LIN {X 0,Y 149.058,Z 383.574,A -85,B 0,C 180,E1 -25603.016,E2 -25603.016} C_VEL
LIN {X 0,Y 150.368,Z 387.947,A -85,B 0,C 180,E1 -25603.742,E2 -25603.742} C_VEL
LIN {X 0,Y 150.892,Z 399.258,A -85,B 0,C 180,E1 -25604.619,E2 -25604.619} C_VEL
LIN {X 0,Y 148.093,Z 440.283,A -85,B 0,C 180,E1 -25606.367,E2 -25606.367} C_VEL
LIN {X 0,Y 146.164,Z 454.102,A -85,B 0,C 180,E1 -25607.428,E2 -25607.428} C_VEL
LIN {X 0,Y 143.596,Z 466.563,A -85,B 0,C 180,E1 -25608.88,E2 -25608.88} C_VEL
LIN {X 0,Y 140.912,Z 476.802,A -85,B 0,C 180,E1 -25610.515,E2 -25610.515} C_VEL
LIN {X 0,Y 137.697,Z 487.195,A -85,B 0,C 180,E1 -25612.695,E2 -25612.695} C_VEL
LIN {X 0,Y 134.338,Z 496.866,A -85,B 0,C 180,E1 -25615.327,E2 -25615.327} C_VEL
LIN {X 0,Y 131.02,Z 505.835,A -85,B 0,C 180,E1 -25618.469,E2 -25618.469} C_VEL
LIN {X 0,Y 127.707,Z 513.721,A -85,B 0,C 180,E1 -25621.923,E2 -25621.923} C_VEL
LIN {X 0,Y 125.501,Z 519.623,A -85,B 0,C 180,E1 -25625.168,E2 -25625.168} C_VEL
LIN {X 0,Y 122.78,Z 526.537,A -85,B 0,C 180,E1 -25629.915,E2 -25629.915} C_VEL
LIN {X 0,Y 120.837,Z 532.058,A -85,B 0,C 180,E1 -25634.83,E2 -25634.83} C_VEL
LIN {X 0,Y 119.81,Z 536.375,A -85,B 0,C 180,E1 -25639.866,E2 -25639.866} C_VEL
LIN {X 0,Y 119.472,Z 538.652,A -85,B 0,C 180,E1 -25643.245,E2 -25643.245} C_VEL
LIN {X 0,Y 119.372,Z 540.456,A -85,B 0,C 180,E1 -25646.627,E2 -25646.627} C_VEL
LIN {X 0,Y 119.478,Z 541.86,A -85,B 0,C 180,E1 -25650.172,E2 -25650.172} C_VEL
LIN {X 0,Y 119.353,Z 542.729,A -85,B 0,C 180,E1 -25653.377,E2 -25653.377} C_VEL
LIN {X 0,Y 119.418,Z 543.262,A -85,B 0,C 180,E1 -25656.761,E2 -25656.761} C_VEL
LIN {X 0,Y 119.832,Z 543.392,A -85,B 0,C 180,E1 -25660.135,E2 -25660.135} C_VEL
LIN {X 0,Y 121.629,Z 542.443,A -85,B 0,C 180,E1 -25666.794,E2 -25666.794} C_VEL
LIN {X 0,Y 123.064,Z 541.401,A -85,B 0,C 180,E1 -25670.04,E2 -25670.04} C_VEL
LIN {X 0,Y 126.605,Z 538.614,A -85,B 0,C 180,E1 -25675.353,E2 -25675.353} C_VEL
LIN {X 0,Y 129.964,Z 535.757,A -85,B 0,C 180,E1 -25679.125,E2 -25679.125} C_VEL
LIN {X 0,Y 134.618,Z 531.251,A -85,B 0,C 180,E1 -25683.418,E2 -25683.418} C_VEL
LIN {X 0,Y 138.6,Z 526.986,A -85,B 0,C 180,E1 -25686.503,E2 -25686.503} C_VEL
LIN {X 0,Y 140.715,Z 524.056,A -85,B 0,C 180,E1 -25688.426,E2 -25688.426} C_VEL
LIN {X 0,Y 142.976,Z 518.943,A -85,B 0,C 180,E1 -25691.745,E2 -25691.745} C_VEL
LIN {X 0,Y 145.492,Z 513.259,A -85,B 0,C 180,E1 -25694.806,E2 -25694.806} C_VEL
LIN {X 0,Y 147.901,Z 509.417,A -85,B 0,C 180,E1 -25696.279,E2 -25696.279} C_VEL
LIN {X 0,Y 154.805,Z 499.219,A -85,B 0,C 180,E1 -25699.006,E2 -25699.006} C_VEL
LIN {X 0,Y 159.828,Z 490.367,A -85,B 0,C 180,E1 -25700.807,E2 -25700.807} C_VEL
LIN {X 0,Y 164.4,Z 481.018,A -85,B 0,C 180,E1 -25702.267,E2 -25702.267} C_VEL
LIN {X 0,Y 169.126,Z 469.344,A -85,B 0,C 180,E1 -25703.623,E2 -25703.623} C_VEL
LIN {X 0,Y 173.178,Z 456.095,A -85,B 0,C 180,E1 -25704.732,E2 -25704.732} C_VEL
LIN {X 0,Y 175.889,Z 443.42,A -85,B 0,C 180,E1 -25705.467,E2 -25705.467} C_VEL
LIN {X 0,Y 177.616,Z 429.252,A -85,B 0,C 180,E1 -25705.973,E2 -25705.973} C_VEL
LIN {X 0,Y 178.336,Z 420.642,A -85,B 0,C 180,E1 -25706.258,E2 -25706.258} C_VEL
LIN {X 0,Y 174.777,Z 410.912,A -85,B 0,C 180,E1 -25709.285,E2 -25709.285} C_VEL
LIN {X 0,Y 170.975,Z 401.854,A -85,B 0,C 180,E1 -25712.952,E2 -25712.952} C_VEL
LIN {X 0,Y 168.609,Z 396.773,A -85,B 0,C 180,E1 -25715.583,E2 -25715.583} C_VEL
LIN {X 0,Y 166.432,Z 392.274,A -85,B 0,C 180,E1 -25718.394,E2 -25718.394} C_VEL
LIN {X 0,Y 164.505,Z 389.028,A -85,B 0,C 180,E1 -25721.312,E2 -25721.312} C_VEL
LIN {X 0,Y 162.526,Z 386.151,A -85,B 0,C 180,E1 -25725.122,E2 -25725.122} C_VEL
LIN {X 0,Y 162.034,Z 384.768,A -85,B 0,C 180,E1 -25726.518,E2 -25726.518} C_VEL
LIN {X 0,Y 160.404,Z 383.082,A -85,B 0,C 180,E1 -25733.431,E2 -25733.431} C_VEL
LIN {X 0,Y 160.639,Z 382.941,A -85,B 0,C 180,E1 -25738.746,E2 -25738.746} C_VEL
LIN {X 0,Y 162.248,Z 384.816,A -85,B 0,C 180,E1 -25744.521,E2 -25744.521} C_VEL
LIN {X 0,Y 163.939,Z 388.212,A -85,B 0,C 180,E1 -25748.271,E2 -25748.271} C_VEL
LIN {X 0,Y 164.958,Z 389.595,A -85,B 0,C 180,E1 -25749.949,E2 -25749.949} C_VEL
LIN {X 0,Y 167.66,Z 394.12,A -85,B 0,C 180,E1 -25753.715,E2 -25753.715} C_VEL
LIN {X 0,Y 170.258,Z 398.497,A -85,B 0,C 180,E1 -25756.64,E2 -25756.64} C_VEL
LIN {X 0,Y 173.134,Z 403.391,A -85,B 0,C 180,E1 -25759.411,E2 -25759.411} C_VEL
LIN {X 0,Y 177.436,Z 411.732,A -85,B 0,C 180,E1 -25763.025,E2 -25763.025} C_VEL
LIN {X 0,Y 178.8,Z 414.577,A -85,B 0,C 180,E1 -25764.067,E2 -25764.067} C_VEL
LIN {X 0,Y 176.796,Z 434.165,A -85,B 0,C 180,E1 -25764.728,E2 -25764.728} C_VEL
LIN {X 0,Y 174.585,Z 446.23,A -85,B 0,C 180,E1 -25765.419,E2 -25765.419} C_VEL
LIN {X 0,Y 171.577,Z 457.31,A -85,B 0,C 180,E1 -25766.265,E2 -25766.265} C_VEL
LIN {X 0,Y 167.687,Z 468.926,A -85,B 0,C 180,E1 -25767.613,E2 -25767.613} C_VEL
LIN {X 0,Y 162.984,Z 479.606,A -85,B 0,C 180,E1 -25769.167,E2 -25769.167} C_VEL
LIN {X 0,Y 157.343,Z 490.399,A -85,B 0,C 180,E1 -25771.322,E2 -25771.322} C_VEL
LIN {X 0,Y 151.116,Z 500.294,A -85,B 0,C 180,E1 -25773.923,E2 -25773.923} C_VEL
LIN {X 0,Y 144.848,Z 508.604,A -85,B 0,C 180,E1 -25776.813,E2 -25776.813} C_VEL
LIN {X 0,Y 138.384,Z 516.119,A -85,B 0,C 180,E1 -25780.376,E2 -25780.376} C_VEL
LIN {X 0,Y 132.495,Z 522.113,A -85,B 0,C 180,E1 -25784.266,E2 -25784.266} C_VEL
LIN {X 0,Y 127.231,Z 526.808,A -85,B 0,C 180,E1 -25788.48,E2 -25788.48} C_VEL
LIN {X 0,Y 122.221,Z 530.713,A -85,B 0,C 180,E1 -25793.613,E2 -25793.613} C_VEL
LIN {X 0,Y 118.941,Z 532.846,A -85,B 0,C 180,E1 -25797.872,E2 -25797.872} C_VEL
LIN {X 0,Y 116.872,Z 533.975,A -85,B 0,C 180,E1 -25801.243,E2 -25801.243} C_VEL
LIN {X 0,Y 113.924,Z 534.95,A -85,B 0,C 180,E1 -25808.274,E2 -25808.274} C_VEL
LIN {X 0,Y 112.953,Z 534.852,A -85,B 0,C 180,E1 -25811.873,E2 -25811.873} C_VEL
LIN {X 0,Y 112.312,Z 534.327,A -85,B 0,C 180,E1 -25815.503,E2 -25815.503} C_VEL
LIN {X 0,Y 112.071,Z 533.382,A -85,B 0,C 180,E1 -25819.154,E2 -25819.154} C_VEL
LIN {X 0,Y 112.159,Z 532.044,A -85,B 0,C 180,E1 -25822.799,E2 -25822.799} C_VEL
LIN {X 0,Y 112.759,Z 529.463,A -85,B 0,C 180,E1 -25827.831,E2 -25827.831} C_VEL
LIN {X 0,Y 113.913,Z 525.425,A -85,B 0,C 180,E1 -25833.535,E2 -25833.535} C_VEL
LIN {X 0,Y 115.858,Z 520.489,A -85,B 0,C 180,E1 -25838.721,E2 -25838.721} C_VEL
LIN {X 0,Y 118.494,Z 514.292,A -85,B 0,C 180,E1 -25843.722,E2 -25843.722} C_VEL
LIN {X 0,Y 121.887,Z 506.562,A -85,B 0,C 180,E1 -25848.487,E2 -25848.487} C_VEL
LIN {X 0,Y 126,Z 496.881,A -85,B 0,C 180,E1 -25852.98,E2 -25852.98} C_VEL
LIN {X 0,Y 129.987,Z 486.863,A -85,B 0,C 180,E1 -25856.489,E2 -25856.489} C_VEL
LIN {X 0,Y 134.034,Z 475.483,A -85,B 0,C 180,E1 -25859.442,E2 -25859.442} C_VEL
LIN {X 0,Y 137.352,Z 464.338,A -85,B 0,C 180,E1 -25861.63,E2 -25861.63} C_VEL
LIN {X 0,Y 139.997,Z 452,A -85,B 0,C 180,E1 -25863.517,E2 -25863.517} C_VEL
LIN {X 0,Y 141.902,Z 439.97,A -85,B 0,C 180,E1 -25864.799,E2 -25864.799} C_VEL
LIN {X 0,Y 143.526,Z 426.582,A -85,B 0,C 180,E1 -25865.609,E2 -25865.609} C_VEL
LIN {X 0,Y 146.26,Z 386.175,A -85,B 0,C 180,E1 -25867.309,E2 -25867.309} C_VEL
LIN {X 0,Y 141.15,Z 375.197,A -85,B 0,C 180,E1 -25870.058,E2 -25870.058} C_VEL
LIN {X 0,Y 136.174,Z 366.246,A -85,B 0,C 180,E1 -25872.941,E2 -25872.941} C_VEL
LIN {X 0,Y 131.196,Z 358.517,A -85,B 0,C 180,E1 -25876.129,E2 -25876.129} C_VEL
LIN {X 0,Y 128.748,Z 355.059,A -85,B 0,C 180,E1 -25877.845,E2 -25877.845} C_VEL
LIN {X 0,Y 125.996,Z 351.155,A -85,B 0,C 180,E1 -25879.951,E2 -25879.951} C_VEL
LIN {X 0,Y 123.491,Z 347.657,A -85,B 0,C 180,E1 -25882.052,E2 -25882.052} C_VEL
LIN {X 0,Y 122.516,Z 346.611,A -85,B 0,C 180,E1 -25882.893,E2 -25882.893} C_VEL
LIN {X 0,Y 120.143,Z 343.788,A -85,B 0,C 180,E1 -25885.123,E2 -25885.123} C_VEL
LIN {X 0,Y 119.192,Z 341.849,A -85,B 0,C 180,E1 -25886.187,E2 -25886.187} C_VEL
LIN {X 0,Y 116.758,Z 340.164,A -85,B 0,C 180,E1 -25888.72,E2 -25888.72} C_VEL
LIN {X 0,Y 115.182,Z 337.57,A -85,B 0,C 180,E1 -25890.783,E2 -25890.783} C_VEL
LIN {X 0,Y 114.864,Z 336.148,A -85,B 0,C 180,E1 -25891.445,E2 -25891.445} C_VEL
LIN {X 0,Y 114.969,Z 336.131,A -85,B 0,C 180,E1 -25898.484,E2 -25898.484} C_VEL
LIN {X 0,Y 115.125,Z 336.141,A -85,B 0,C 180,E1 -25905.867,E2 -25905.867} C_VEL
LIN {X 0,Y 115.315,Z 336.084,A -85,B 0,C 180,E1 -25909.465,E2 -25909.465} C_VEL
LIN {X 0,Y 115.512,Z 336.092,A -85,B 0,C 180,E1 -25916.512,E2 -25916.512} C_VEL
LIN {X 0,Y 115.986,Z 336,A -85,B 0,C 180,E1 -25920,E2 -25920} C_VEL
LIN {X 0,Y 115.382,Z 336.107,A -85,B 0,C 180,E1 -25926.998,E2 -25926.998} C_VEL
LIN {X 0,Y 115.28,Z 336.096,A -85,B 0,C 180,E1 -25932.738,E2 -25932.738} C_VEL
LIN {X 0,Y 114.982,Z 336.156,A -85,B 0,C 180,E1 -25938.256,E2 -25938.256} C_VEL
LIN {X 0,Y 115.679,Z 338.437,A -85,B 0,C 180,E1 -25939.406,E2 -25939.406} C_VEL
LIN {X 0,Y 117.509,Z 340.782,A -85,B 0,C 180,E1 -25941.614,E2 -25941.614} C_VEL
LIN {X 0,Y 119.474,Z 342.161,A -85,B 0,C 180,E1 -25943.604,E2 -25943.604} C_VEL
LIN {X 0,Y 121.215,Z 345.242,A -85,B 0,C 180,E1 -25945.431,E2 -25945.431} C_VEL
LIN {X 0,Y 123.493,Z 347.501,A -85,B 0,C 180,E1 -25947.428,E2 -25947.428} C_VEL
LIN {X 0,Y 125.957,Z 351.004,A -85,B 0,C 180,E1 -25949.504,E2 -25949.504} C_VEL
LIN {X 0,Y 127.235,Z 352.704,A -85,B 0,C 180,E1 -25950.497,E2 -25950.497} C_VEL
LIN {X 0,Y 130.55,Z 357.466,A -85,B 0,C 180,E1 -25952.915,E2 -25952.915} C_VEL
LIN {X 0,Y 135.628,Z 365.423,A -85,B 0,C 180,E1 -25956.232,E2 -25956.232} C_VEL
LIN {X 0,Y 140.635,Z 376.726,A -85,B 0,C 180,E1 -25959.335,E2 -25959.335} C_VEL
LIN {X 0,Y 144.693,Z 388.412,A -85,B 0,C 180,E1 -25961.757,E2 -25961.757} C_VEL
LIN {X 0,Y 145.243,Z 391.387,A -85,B 0,C 180,E1 -25962.161,E2 -25962.161} C_VEL
LIN {X 0,Y 145.524,Z 400.032,A -85,B 0,C 180,E1 -25962.835,E2 -25962.835} C_VEL
LIN {X 0,Y 142.651,Z 440.166,A -85,B 0,C 180,E1 -25964.583,E2 -25964.583} C_VEL
LIN {X 0,Y 140.679,Z 453.603,A -85,B 0,C 180,E1 -25965.624,E2 -25965.624} C_VEL
LIN {X 0,Y 138.048,Z 466.019,A -85,B 0,C 180,E1 -25967.087,E2 -25967.087} C_VEL
LIN {X 0,Y 134.981,Z 477.113,A -85,B 0,C 180,E1 -25968.906,E2 -25968.906} C_VEL
LIN {X 0,Y 131.619,Z 487.401,A -85,B 0,C 180,E1 -25971.144,E2 -25971.144} C_VEL
LIN {X 0,Y 128.101,Z 496.992,A -85,B 0,C 180,E1 -25973.861,E2 -25973.861} C_VEL
LIN {X 0,Y 124.234,Z 506.798,A -85,B 0,C 180,E1 -25977.494,E2 -25977.494} C_VEL
LIN {X 0,Y 120.666,Z 515.078,A -85,B 0,C 180,E1 -25981.453,E2 -25981.453} C_VEL
LIN {X 0,Y 117.508,Z 522.647,A -85,B 0,C 180,E1 -25986.192,E2 -25986.192} C_VEL
LIN {X 0,Y 115.266,Z 527.977,A -85,B 0,C 180,E1 -25990.409,E2 -25990.409} C_VEL
LIN {X 0,Y 113.469,Z 533.142,A -85,B 0,C 180,E1 -25995.658,E2 -25995.658} C_VEL
LIN {X 0,Y 112.552,Z 537.14,A -85,B 0,C 180,E1 -26001.021,E2 -26001.021} C_VEL
LIN {X 0,Y 112.275,Z 540.071,A -85,B 0,C 180,E1 -26006.413,E2 -26006.413} C_VEL
LIN {X 0,Y 112.41,Z 541.451,A -85,B 0,C 180,E1 -26010.002,E2 -26010.002} C_VEL
LIN {X 0,Y 112.262,Z 542.4,A -85,B 0,C 180,E1 -26013.591,E2 -26013.591} C_VEL
LIN {X 0,Y 112.815,Z 543.13,A -85,B 0,C 180,E1 -26020.773,E2 -26020.773} C_VEL
LIN {X 0,Y 114.804,Z 542.241,A -85,B 0,C 180,E1 -26027.825,E2 -26027.825} C_VEL
LIN {X 0,Y 116.397,Z 541.225,A -85,B 0,C 180,E1 -26031.242,E2 -26031.242} C_VEL
LIN {X 0,Y 118.505,Z 539.825,A -85,B 0,C 180,E1 -26034.53,E2 -26034.53} C_VEL
LIN {X 0,Y 122.316,Z 536.898,A -85,B 0,C 180,E1 -26039.236,E2 -26039.236} C_VEL
LIN {X 0,Y 127.787,Z 532.129,A -85,B 0,C 180,E1 -26044.414,E2 -26044.414} C_VEL
LIN {X 0,Y 134.001,Z 525.957,A -85,B 0,C 180,E1 -26049.005,E2 -26049.005} C_VEL
LIN {X 0,Y 140.224,Z 519.174,A -85,B 0,C 180,E1 -26052.581,E2 -26052.581} C_VEL
LIN {X 0,Y 146.925,Z 510.774,A -85,B 0,C 180,E1 -26055.85,E2 -26055.85} C_VEL
LIN {X 0,Y 147.901,Z 509.417,A -85,B 0,C 180,E1 -26056.279,E2 -26056.279} C_VEL
LIN {X 0,Y 149.337,Z 506.782,A -85,B 0,C 180,E1 -26057.292,E2 -26057.292} C_VEL
LIN {X 0,Y 151.415,Z 498.223,A -85,B 0,C 180,E1 -26061.216,E2 -26061.216} C_VEL
LIN {X 0,Y 152.916,Z 495.22,A -85,B 0,C 180,E1 -26062.02,E2 -26062.02} C_VEL
LIN {X 0,Y 158.797,Z 484.534,A -85,B 0,C 180,E1 -26063.874,E2 -26063.874} C_VEL
LIN {X 0,Y 164.353,Z 472.099,A -85,B 0,C 180,E1 -26065.404,E2 -26065.404} C_VEL
LIN {X 0,Y 168.557,Z 459.912,A -85,B 0,C 180,E1 -26066.502,E2 -26066.502} C_VEL
LIN {X 0,Y 171.647,Z 447.32,A -85,B 0,C 180,E1 -26067.32,E2 -26067.32} C_VEL
LIN {X 0,Y 173.74,Z 434.201,A -85,B 0,C 180,E1 -26067.837,E2 -26067.837} C_VEL
LIN {X 0,Y 174.69,Z 423.526,A -85,B 0,C 180,E1 -26068.209,E2 -26068.209} C_VEL
LIN {X 0,Y 171.782,Z 415.209,A -85,B 0,C 180,E1 -26070.958,E2 -26070.958} C_VEL
LIN {X 0,Y 168.456,Z 406.824,A -85,B 0,C 180,E1 -26074.517,E2 -26074.517} C_VEL
LIN {X 0,Y 166.429,Z 402.301,A -85,B 0,C 180,E1 -26077.007,E2 -26077.007} C_VEL
LIN {X 0,Y 164.818,Z 398.66,A -85,B 0,C 180,E1 -26079.313,E2 -26079.313} C_VEL
LIN {X 0,Y 163.102,Z 395.672,A -85,B 0,C 180,E1 -26082.116,E2 -26082.116} C_VEL
LIN {X 0,Y 161.287,Z 392.716,A -85,B 0,C 180,E1 -26085.972,E2 -26085.972} C_VEL
LIN {X 0,Y 160.824,Z 391.582,A -85,B 0,C 180,E1 -26087.379,E2 -26087.379} C_VEL
LIN {X 0,Y 159.535,Z 390.137,A -85,B 0,C 180,E1 -26093.395,E2 -26093.395} C_VEL
LIN {X 0,Y 159.763,Z 390.006,A -85,B 0,C 180,E1 -26098.739,E2 -26098.739} C_VEL
LIN {X 0,Y 161.135,Z 391.709,A -85,B 0,C 180,E1 -26103.964,E2 -26103.964} C_VEL
LIN {X 0,Y 162.856,Z 395.183,A -85,B 0,C 180,E1 -26107.966,E2 -26107.966} C_VEL
LIN {X 0,Y 163.772,Z 396.681,A -85,B 0,C 180,E1 -26109.572,E2 -26109.572} C_VEL
LIN {X 0,Y 165.944,Z 400.463,A -85,B 0,C 180,E1 -26112.788,E2 -26112.788} C_VEL
LIN {X 0,Y 168.585,Z 405.148,A -85,B 0,C 180,E1 -26115.955,E2 -26115.955} C_VEL
LIN {X 0,Y 171.805,Z 411.108,A -85,B 0,C 180,E1 -26119.204,E2 -26119.204} C_VEL
LIN {X 0,Y 175.138,Z 418.033,A -85,B 0,C 180,E1 -26122.142,E2 -26122.142} C_VEL
LIN {X 0,Y 173.251,Z 435.224,A -85,B 0,C 180,E1 -26122.74,E2 -26122.74} C_VEL
LIN {X 0,Y 170.677,Z 448.21,A -85,B 0,C 180,E1 -26123.49,E2 -26123.49} C_VEL
LIN {X 0,Y 167.095,Z 460.345,A -85,B 0,C 180,E1 -26124.485,E2 -26124.485} C_VEL
LIN {X 0,Y 162.984,Z 471.437,A -85,B 0,C 180,E1 -26125.821,E2 -26125.821} C_VEL
LIN {X 0,Y 158.247,Z 481.527,A -85,B 0,C 180,E1 -26127.346,E2 -26127.346} C_VEL
LIN {X 0,Y 152.41,Z 492.029,A -85,B 0,C 180,E1 -26129.497,E2 -26129.497} C_VEL
LIN {X 0,Y 145.675,Z 501.926,A -85,B 0,C 180,E1 -26132.186,E2 -26132.186} C_VEL
LIN {X 0,Y 139.44,Z 509.733,A -85,B 0,C 180,E1 -26135.011,E2 -26135.011} C_VEL
LIN {X 0,Y 132.701,Z 517.096,A -85,B 0,C 180,E1 -26138.63,E2 -26138.63} C_VEL
LIN {X 0,Y 127.444,Z 522.101,A -85,B 0,C 180,E1 -26141.966,E2 -26141.966} C_VEL
LIN {X 0,Y 121.858,Z 526.805,A -85,B 0,C 180,E1 -26146.203,E2 -26146.203} C_VEL
LIN {X 0,Y 118.511,Z 529.349,A -85,B 0,C 180,E1 -26149.281,E2 -26149.281} C_VEL
LIN {X 0,Y 115.505,Z 531.376,A -85,B 0,C 180,E1 -26152.52,E2 -26152.52} C_VEL
LIN {X 0,Y 112.833,Z 532.976,A -85,B 0,C 180,E1 -26155.902,E2 -26155.902} C_VEL
LIN {X 0,Y 110.542,Z 534.159,A -85,B 0,C 180,E1 -26159.426,E2 -26159.426} C_VEL
LIN {X 0,Y 107.361,Z 535.189,A -85,B 0,C 180,E1 -26166.413,E2 -26166.413} C_VEL
LIN {X 0,Y 106.08,Z 535.137,A -85,B 0,C 180,E1 -26170.653,E2 -26170.653} C_VEL
LIN {X 0,Y 105.326,Z 534.671,A -85,B 0,C 180,E1 -26174.518,E2 -26174.518} C_VEL
LIN {X 0,Y 104.986,Z 533.76,A -85,B 0,C 180,E1 -26178.413,E2 -26178.413} C_VEL
LIN {X 0,Y 105.029,Z 532.452,A -85,B 0,C 180,E1 -26182.307,E2 -26182.307} C_VEL
LIN {X 0,Y 105.574,Z 530.372,A -85,B 0,C 180,E1 -26186.896,E2 -26186.896} C_VEL
LIN {X 0,Y 106.833,Z 525.96,A -85,B 0,C 180,E1 -26193.77,E2 -26193.77} C_VEL
LIN {X 0,Y 108.855,Z 521.097,A -85,B 0,C 180,E1 -26199.286,E2 -26199.286} C_VEL
LIN {X 0,Y 111.636,Z 514.979,A -85,B 0,C 180,E1 -26204.583,E2 -26204.583} C_VEL
LIN {X 0,Y 115.203,Z 507.379,A -85,B 0,C 180,E1 -26209.602,E2 -26209.602} C_VEL
LIN {X 0,Y 118.774,Z 499.595,A -85,B 0,C 180,E1 -26213.539,E2 -26213.539} C_VEL
LIN {X 0,Y 123.272,Z 489.019,A -85,B 0,C 180,E1 -26217.593,E2 -26217.593} C_VEL
LIN {X 0,Y 127.364,Z 478.243,A -85,B 0,C 180,E1 -26220.689,E2 -26220.689} C_VEL
LIN {X 0,Y 130.893,Z 467.702,A -85,B 0,C 180,E1 -26222.929,E2 -26222.929} C_VEL
LIN {X 0,Y 133.759,Z 456.244,A -85,B 0,C 180,E1 -26224.845,E2 -26224.845} C_VEL
LIN {X 0,Y 136.162,Z 442.69,A -85,B 0,C 180,E1 -26226.516,E2 -26226.516} C_VEL
LIN {X 0,Y 137.952,Z 430.118,A -85,B 0,C 180,E1 -26227.385,E2 -26227.385} C_VEL
LIN {X 0,Y 141.014,Z 388.433,A -85,B 0,C 180,E1 -26229.17,E2 -26229.17} C_VEL
LIN {X 0,Y 135.998,Z 377.744,A -85,B 0,C 180,E1 -26232.128,E2 -26232.128} C_VEL
LIN {X 0,Y 131.738,Z 370.125,A -85,B 0,C 180,E1 -26234.842,E2 -26234.842} C_VEL
LIN {X 0,Y 126.521,Z 361.692,A -85,B 0,C 180,E1 -26238.587,E2 -26238.587} C_VEL
LIN {X 0,Y 122.815,Z 356.611,A -85,B 0,C 180,E1 -26241.588,E2 -26241.588} C_VEL
LIN {X 0,Y 120.2,Z 352.921,A -85,B 0,C 180,E1 -26243.997,E2 -26243.997} C_VEL
LIN {X 0,Y 117.668,Z 349.729,A -85,B 0,C 180,E1 -26246.567,E2 -26246.567} C_VEL
LIN {X 0,Y 116.821,Z 348.305,A -85,B 0,C 180,E1 -26247.549,E2 -26247.549} C_VEL
LIN {X 0,Y 114.278,Z 345.935,A -85,B 0,C 180,E1 -26250.529,E2 -26250.529} C_VEL
LIN {X 0,Y 112.719,Z 342.91,A -85,B 0,C 180,E1 -26252.876,E2 -26252.876} C_VEL
LIN {X 0,Y 110.02,Z 341.269,A -85,B 0,C 180,E1 -26257.078,E2 -26257.078} C_VEL
LIN {X 0,Y 108.256,Z 338.534,A -85,B 0,C 180,E1 -26261.059,E2 -26261.059} C_VEL
LIN {X 0,Y 107.951,Z 337.013,A -85,B 0,C 180,E1 -26262.232,E2 -26262.232} C_VEL
LIN {X 0,Y 108.244,Z 336.966,A -85,B 0,C 180,E1 -26268.768,E2 -26268.768} C_VEL
LIN {X 0,Y 108.436,Z 336.974,A -85,B 0,C 180,E1 -26276.284,E2 -26276.284} C_VEL
LIN {X 0,Y 108.912,Z 336.88,A -85,B 0,C 180,E1 -26280,E2 -26280} C_VEL
LIN {X 0,Y 108.307,Z 337.14,A -85,B 0,C 180,E1 -26288.161,E2 -26288.161} C_VEL
LIN {X 0,Y 108.93,Z 339.134,A -85,B 0,C 180,E1 -26289.986,E2 -26289.986} C_VEL
LIN {X 0,Y 111.133,Z 342.004,A -85,B 0,C 180,E1 -26294.294,E2 -26294.294} C_VEL
LIN {X 0,Y 112.956,Z 343.095,A -85,B 0,C 180,E1 -26296.957,E2 -26296.957} C_VEL
LIN {X 0,Y 114.67,Z 346.299,A -85,B 0,C 180,E1 -26299.467,E2 -26299.467} C_VEL
LIN {X 0,Y 117.199,Z 348.643,A -85,B 0,C 180,E1 -26302.36,E2 -26302.36} C_VEL
LIN {X 0,Y 119.447,Z 352.116,A -85,B 0,C 180,E1 -26304.786,E2 -26304.786} C_VEL
LIN {X 0,Y 121.018,Z 353.847,A -85,B 0,C 180,E1 -26306.255,E2 -26306.255} C_VEL
LIN {X 0,Y 124.747,Z 359.196,A -85,B 0,C 180,E1 -26309.516,E2 -26309.516} C_VEL
LIN {X 0,Y 128.743,Z 365.107,A -85,B 0,C 180,E1 -26312.563,E2 -26312.563} C_VEL
LIN {X 0,Y 132.484,Z 371.714,A -85,B 0,C 180,E1 -26315.175,E2 -26315.175} C_VEL
LIN {X 0,Y 136.515,Z 381.439,A -85,B 0,C 180,E1 -26317.891,E2 -26317.891} C_VEL
LIN {X 0,Y 140.078,Z 392.284,A -85,B 0,C 180,E1 -26320.22,E2 -26320.22} C_VEL
LIN {X 0,Y 140.289,Z 401.392,A -85,B 0,C 180,E1 -26320.95,E2 -26320.95} C_VEL
LIN {X 0,Y 137.408,Z 439.493,A -85,B 0,C 180,E1 -26322.619,E2 -26322.619} C_VEL
LIN {X 0,Y 135.385,Z 452.908,A -85,B 0,C 180,E1 -26323.658,E2 -26323.658} C_VEL
LIN {X 0,Y 132.651,Z 465.467,A -85,B 0,C 180,E1 -26325.148,E2 -26325.148} C_VEL
LIN {X 0,Y 129.167,Z 477.424,A -85,B 0,C 180,E1 -26327.149,E2 -26327.149} C_VEL
LIN {X 0,Y 125.647,Z 487.607,A -85,B 0,C 180,E1 -26329.443,E2 -26329.443} C_VEL
LIN {X 0,Y 121.955,Z 497.117,A -85,B 0,C 180,E1 -26332.247,E2 -26332.247} C_VEL
LIN {X 0,Y 118.264,Z 505.957,A -85,B 0,C 180,E1 -26335.632,E2 -26335.632} C_VEL
LIN {X 0,Y 114.47,Z 513.933,A -85,B 0,C 180,E1 -26339.491,E2 -26339.491} C_VEL
LIN {X 0,Y 112.082,Z 519.544,A -85,B 0,C 180,E1 -26342.963,E2 -26342.963} C_VEL
LIN {X 0,Y 109.011,Z 526.376,A -85,B 0,C 180,E1 -26348.243,E2 -26348.243} C_VEL
LIN {X 0,Y 106.554,Z 532.637,A -85,B 0,C 180,E1 -26354.705,E2 -26354.705} C_VEL
LIN {X 0,Y 105.525,Z 536.695,A -85,B 0,C 180,E1 -26360.418,E2 -26360.418} C_VEL
LIN {X 0,Y 105.192,Z 539.674,A -85,B 0,C 180,E1 -26366.171,E2 -26366.171} C_VEL
LIN {X 0,Y 105.334,Z 541.098,A -85,B 0,C 180,E1 -26370.002,E2 -26370.002} C_VEL
LIN {X 0,Y 105.18,Z 542.071,A -85,B 0,C 180,E1 -26373.833,E2 -26373.833} C_VEL
LIN {X 0,Y 105.829,Z 542.857,A -85,B 0,C 180,E1 -26381.494,E2 -26381.494} C_VEL
LIN {X 0,Y 106.738,Z 542.651,A -85,B 0,C 180,E1 -26385.272,E2 -26385.272} C_VEL
LIN {X 0,Y 109.792,Z 541.049,A -85,B 0,C 180,E1 -26392.588,E2 -26392.588} C_VEL
LIN {X 0,Y 112.069,Z 539.676,A -85,B 0,C 180,E1 -26396.041,E2 -26396.041} C_VEL
LIN {X 0,Y 116.164,Z 536.804,A -85,B 0,C 180,E1 -26400.949,E2 -26400.949} C_VEL
LIN {X 0,Y 121.517,Z 532.511,A -85,B 0,C 180,E1 -26405.933,E2 -26405.933} C_VEL
LIN {X 0,Y 126.534,Z 527.957,A -85,B 0,C 180,E1 -26409.699,E2 -26409.699} C_VEL
LIN {X 0,Y 132.817,Z 521.733,A -85,B 0,C 180,E1 -26413.465,E2 -26413.465} C_VEL
LIN {X 0,Y 139.722,Z 513.99,A -85,B 0,C 180,E1 -26416.833,E2 -26416.833} C_VEL
LIN {X 0,Y 145.785,Z 506.103,A -85,B 0,C 180,E1 -26419.402,E2 -26419.402} C_VEL
LIN {X 0,Y 152.777,Z 495.437,A -85,B 0,C 180,E1 -26421.98,E2 -26421.98} C_VEL
LIN {X 0,Y 152.916,Z 495.22,A -85,B 0,C 180,E1 -26422.02,E2 -26422.02} C_VEL
LIN {X 0,Y 154.432,Z 492.177,A -85,B 0,C 180,E1 -26422.792,E2 -26422.792} C_VEL
LIN {X 0,Y 155.587,Z 487.389,A -85,B 0,C 180,E1 -26424.503,E2 -26424.503} C_VEL
LIN {X 0,Y 156.585,Z 482.399,A -85,B 0,C 180,E1 -26426.148,E2 -26426.148} C_VEL
LIN {X 0,Y 157.789,Z 479.033,A -85,B 0,C 180,E1 -26426.8,E2 -26426.8} C_VEL
LIN {X 0,Y 162.599,Z 467.472,A -85,B 0,C 180,E1 -26428.023,E2 -26428.023} C_VEL
LIN {X 0,Y 166.262,Z 456.038,A -85,B 0,C 180,E1 -26428.921,E2 -26428.921} C_VEL
LIN {X 0,Y 169.27,Z 442.933,A -85,B 0,C 180,E1 -26429.634,E2 -26429.634} C_VEL
LIN {X 0,Y 171.191,Z 427.879,A -85,B 0,C 180,E1 -26430.144,E2 -26430.144} C_VEL
LIN {X 0,Y 171.199,Z 426.272,A -85,B 0,C 180,E1 -26430.294,E2 -26430.294} C_VEL
LIN {X 0,Y 168.682,Z 418.863,A -85,B 0,C 180,E1 -26432.966,E2 -26432.966} C_VEL
LIN {X 0,Y 166.001,Z 411.729,A -85,B 0,C 180,E1 -26436.201,E2 -26436.201} C_VEL
LIN {X 0,Y 164.477,Z 408.103,A -85,B 0,C 180,E1 -26438.292,E2 -26438.292} C_VEL
LIN {X 0,Y 163.248,Z 405.113,A -85,B 0,C 180,E1 -26440.243,E2 -26440.243} C_VEL
LIN {X 0,Y 161.939,Z 402.552,A -85,B 0,C 180,E1 -26442.559,E2 -26442.559} C_VEL
LIN {X 0,Y 160.156,Z 399.511,A -85,B 0,C 180,E1 -26446.599,E2 -26446.599} C_VEL
LIN {X 0,Y 159.75,Z 398.506,A -85,B 0,C 180,E1 -26447.935,E2 -26447.935} C_VEL
LIN {X 0,Y 158.667,Z 397.194,A -85,B 0,C 180,E1 -26453.359,E2 -26453.359} C_VEL
LIN {X 0,Y 158.886,Z 397.086,A -85,B 0,C 180,E1 -26458.732,E2 -26458.732} C_VEL
LIN {X 0,Y 160.057,Z 398.646,A -85,B 0,C 180,E1 -26463.461,E2 -26463.461} C_VEL
LIN {X 0,Y 161.849,Z 402.289,A -85,B 0,C 180,E1 -26467.799,E2 -26467.799} C_VEL
LIN {X 0,Y 164.29,Z 406.842,A -85,B 0,C 180,E1 -26471.859,E2 -26471.859} C_VEL
LIN {X 0,Y 166.732,Z 411.396,A -85,B 0,C 180,E1 -26475.014,E2 -26475.014} C_VEL
LIN {X 0,Y 170.002,Z 417.868,A -85,B 0,C 180,E1 -26478.53,E2 -26478.53} C_VEL
LIN {X 0,Y 171.684,Z 421.513,A -85,B 0,C 180,E1 -26480.142,E2 -26480.142} C_VEL
LIN {X 0,Y 169.828,Z 436.904,A -85,B 0,C 180,E1 -26480.699,E2 -26480.699} C_VEL
LIN {X 0,Y 166.894,Z 450.204,A -85,B 0,C 180,E1 -26481.476,E2 -26481.476} C_VEL
LIN {X 0,Y 163.438,Z 461.342,A -85,B 0,C 180,E1 -26482.405,E2 -26482.405} C_VEL
LIN {X 0,Y 158.556,Z 473.73,A -85,B 0,C 180,E1 -26483.906,E2 -26483.906} C_VEL
LIN {X 0,Y 153.679,Z 483.441,A -85,B 0,C 180,E1 -26485.416,E2 -26485.416} C_VEL
LIN {X 0,Y 148.298,Z 492.561,A -85,B 0,C 180,E1 -26487.303,E2 -26487.303} C_VEL
LIN {X 0,Y 141.271,Z 502.43,A -85,B 0,C 180,E1 -26489.969,E2 -26489.969} C_VEL
LIN {X 0,Y 134.169,Z 510.861,A -85,B 0,C 180,E1 -26493.057,E2 -26493.057} C_VEL
LIN {X 0,Y 127.142,Z 518.045,A -85,B 0,C 180,E1 -26496.723,E2 -26496.723} C_VEL
LIN {X 0,Y 120.676,Z 523.724,A -85,B 0,C 180,E1 -26500.789,E2 -26500.789} C_VEL
LIN {X 0,Y 114.838,Z 528.159,A -85,B 0,C 180,E1 -26505.266,E2 -26505.266} C_VEL
LIN {X 0,Y 109.813,Z 531.477,A -85,B 0,C 180,E1 -26510.206,E2 -26510.206} C_VEL
LIN {X 0,Y 106.881,Z 533.109,A -85,B 0,C 180,E1 -26513.713,E2 -26513.713} C_VEL
LIN {X 0,Y 104.324,Z 534.327,A -85,B 0,C 180,E1 -26517.387,E2 -26517.387} C_VEL
LIN {X 0,Y 102.233,Z 535.108,A -85,B 0,C 180,E1 -26521.233,E2 -26521.233} C_VEL
LIN {X 0,Y 100.496,Z 535.465,A -85,B 0,C 180,E1 -26525.385,E2 -26525.385} C_VEL
LIN {X 0,Y 98.379,Z 534.996,A -85,B 0,C 180,E1 -26533.394,E2 -26533.394} C_VEL
LIN {X 0,Y 97.93,Z 534.136,A -85,B 0,C 180,E1 -26537.565,E2 -26537.565} C_VEL
LIN {X 0,Y 97.9,Z 532.859,A -85,B 0,C 180,E1 -26541.743,E2 -26541.743} C_VEL
LIN {X 0,Y 98.503,Z 530.528,A -85,B 0,C 180,E1 -26547.269,E2 -26547.269} C_VEL
LIN {X 0,Y 99.758,Z 526.493,A -85,B 0,C 180,E1 -26554.038,E2 -26554.038} C_VEL
LIN {X 0,Y 101.862,Z 521.703,A -85,B 0,C 180,E1 -26559.93,E2 -26559.93} C_VEL
LIN {X 0,Y 104.809,Z 515.662,A -85,B 0,C 180,E1 -26565.556,E2 -26565.556} C_VEL
LIN {X 0,Y 108.566,Z 508.157,A -85,B 0,C 180,E1 -26570.855,E2 -26570.855} C_VEL
LIN {X 0,Y 112.302,Z 500.493,A -85,B 0,C 180,E1 -26574.985,E2 -26574.985} C_VEL
LIN {X 0,Y 116.608,Z 491.147,A -85,B 0,C 180,E1 -26578.824,E2 -26578.824} C_VEL
LIN {X 0,Y 120.863,Z 480.759,A -85,B 0,C 180,E1 -26582.044,E2 -26582.044} C_VEL
LIN {X 0,Y 125.021,Z 469.195,A -85,B 0,C 180,E1 -26584.69,E2 -26584.69} C_VEL
LIN {X 0,Y 128.303,Z 457.058,A -85,B 0,C 180,E1 -26586.804,E2 -26586.804} C_VEL
LIN {X 0,Y 130.838,Z 443.723,A -85,B 0,C 180,E1 -26588.502,E2 -26588.502} C_VEL
LIN {X 0,Y 132.779,Z 430.91,A -85,B 0,C 180,E1 -26589.429,E2 -26589.429} C_VEL
LIN {X 0,Y 135.911,Z 390.91,A -85,B 0,C 180,E1 -26591.158,E2 -26591.158} C_VEL
LIN {X 0,Y 131.469,Z 381.245,A -85,B 0,C 180,E1 -26594.05,E2 -26594.05} C_VEL
LIN {X 0,Y 126.95,Z 373.1,A -85,B 0,C 180,E1 -26597.254,E2 -26597.254} C_VEL
LIN {X 0,Y 122.921,Z 366.648,A -85,B 0,C 180,E1 -26600.463,E2 -26600.463} C_VEL
LIN {X 0,Y 119.927,Z 362.246,A -85,B 0,C 180,E1 -26603.144,E2 -26603.144} C_VEL
LIN {X 0,Y 117.808,Z 359.09,A -85,B 0,C 180,E1 -26605.268,E2 -26605.268} C_VEL
LIN {X 0,Y 115.239,Z 355.619,A -85,B 0,C 180,E1 -26608.11,E2 -26608.11} C_VEL
LIN {X 0,Y 114.497,Z 354.56,A -85,B 0,C 180,E1 -26609.018,E2 -26609.018} C_VEL
LIN {X 0,Y 112.066,Z 351.854,A -85,B 0,C 180,E1 -26612.198,E2 -26612.198} C_VEL
LIN {X 0,Y 110.943,Z 349.671,A -85,B 0,C 180,E1 -26614.043,E2 -26614.043} C_VEL
LIN {X 0,Y 108.321,Z 347.658,A -85,B 0,C 180,E1 -26618.596,E2 -26618.596} C_VEL
LIN {X 0,Y 106.783,Z 344.806,A -85,B 0,C 180,E1 -26622.649,E2 -26622.649} C_VEL
LIN {X 0,Y 106.487,Z 343.968,A -85,B 0,C 180,E1 -26623.711,E2 -26623.711} C_VEL
LIN {X 0,Y 104.687,Z 342.995,A -85,B 0,C 180,E1 -26636.151,E2 -26636.151} C_VEL
LIN {X 0,Y 105.277,Z 343.114,A -85,B 0,C 180,E1 -26641.074,E2 -26641.074} C_VEL
LIN {X 0,Y 106.958,Z 344.145,A -85,B 0,C 180,E1 -26647.077,E2 -26647.077} C_VEL
LIN {X 0,Y 108.408,Z 347.309,A -85,B 0,C 180,E1 -26650.979,E2 -26650.979} C_VEL
LIN {X 0,Y 110.764,Z 349.493,A -85,B 0,C 180,E1 -26655.173,E2 -26655.173} C_VEL
LIN {X 0,Y 111.303,Z 350.189,A -85,B 0,C 180,E1 -26656.037,E2 -26656.037} C_VEL
LIN {X 0,Y 113.459,Z 353.545,A -85,B 0,C 180,E1 -26659.213,E2 -26659.213} C_VEL
LIN {X 0,Y 115.12,Z 355.247,A -85,B 0,C 180,E1 -26661.224,E2 -26661.224} C_VEL
LIN {X 0,Y 117.587,Z 358.821,A -85,B 0,C 180,E1 -26664.007,E2 -26664.007} C_VEL
LIN {X 0,Y 118.744,Z 360.345,A -85,B 0,C 180,E1 -26665.177,E2 -26665.177} C_VEL
LIN {X 0,Y 121.923,Z 365.052,A -85,B 0,C 180,E1 -26668.161,E2 -26668.161} C_VEL
LIN {X 0,Y 125.574,Z 370.719,A -85,B 0,C 180,E1 -26671.178,E2 -26671.178} C_VEL
LIN {X 0,Y 128.6,Z 376.257,A -85,B 0,C 180,E1 -26673.479,E2 -26673.479} C_VEL
LIN {X 0,Y 132.301,Z 385.659,A -85,B 0,C 180,E1 -26676.227,E2 -26676.227} C_VEL
LIN {X 0,Y 135.162,Z 394.739,A -85,B 0,C 180,E1 -26678.295,E2 -26678.295} C_VEL
LIN {X 0,Y 135.32,Z 400.861,A -85,B 0,C 180,E1 -26678.83,E2 -26678.83} C_VEL
LIN {X 0,Y 132.264,Z 439.412,A -85,B 0,C 180,E1 -26680.544,E2 -26680.544} C_VEL
LIN {X 0,Y 130.118,Z 452.95,A -85,B 0,C 180,E1 -26681.609,E2 -26681.609} C_VEL
LIN {X 0,Y 127.421,Z 464.886,A -85,B 0,C 180,E1 -26683.049,E2 -26683.049} C_VEL
LIN {X 0,Y 124.056,Z 476.135,A -85,B 0,C 180,E1 -26684.919,E2 -26684.919} C_VEL
LIN {X 0,Y 119.795,Z 487.804,A -85,B 0,C 180,E1 -26687.575,E2 -26687.575} C_VEL
LIN {X 0,Y 115.917,Z 497.238,A -85,B 0,C 180,E1 -26690.464,E2 -26690.464} C_VEL
LIN {X 0,Y 111.601,Z 506.916,A -85,B 0,C 180,E1 -26694.376,E2 -26694.376} C_VEL
LIN {X 0,Y 107.666,Z 514.807,A -85,B 0,C 180,E1 -26698.522,E2 -26698.522} C_VEL
LIN {X 0,Y 104.523,Z 521.372,A -85,B 0,C 180,E1 -26703.011,E2 -26703.011} C_VEL
LIN {X 0,Y 101.917,Z 526.805,A -85,B 0,C 180,E1 -26707.714,E2 -26707.714} C_VEL
LIN {X 0,Y 99.686,Z 532.116,A -85,B 0,C 180,E1 -26713.623,E2 -26713.623} C_VEL
LIN {X 0,Y 98.501,Z 536.235,A -85,B 0,C 180,E1 -26719.727,E2 -26719.727} C_VEL
LIN {X 0,Y 98.101,Z 539.266,A -85,B 0,C 180,E1 -26725.894,E2 -26725.894} C_VEL
LIN {X 0,Y 98.245,Z 540.744,A -85,B 0,C 180,E1 -26730.002,E2 -26730.002} C_VEL
LIN {X 0,Y 98.091,Z 541.742,A -85,B 0,C 180,E1 -26734.111,E2 -26734.111} C_VEL
LIN {X 0,Y 98.872,Z 542.579,A -85,B 0,C 180,E1 -26742.315,E2 -26742.315} C_VEL
LIN {X 0,Y 99.863,Z 542.419,A -85,B 0,C 180,E1 -26746.352,E2 -26746.352} C_VEL
LIN {X 0,Y 103.261,Z 540.876,A -85,B 0,C 180,E1 -26754.104,E2 -26754.104} C_VEL
LIN {X 0,Y 108.525,Z 537.783,A -85,B 0,C 180,E1 -26761.205,E2 -26761.205} C_VEL
LIN {X 0,Y 114.242,Z 533.721,A -85,B 0,C 180,E1 -26766.698,E2 -26766.698} C_VEL
LIN {X 0,Y 121.154,Z 527.991,A -85,B 0,C 180,E1 -26771.845,E2 -26771.845} C_VEL
LIN {X 0,Y 127.766,Z 521.837,A -85,B 0,C 180,E1 -26775.652,E2 -26775.652} C_VEL
LIN {X 0,Y 134.963,Z 514.207,A -85,B 0,C 180,E1 -26779.033,E2 -26779.033} C_VEL
LIN {X 0,Y 141.283,Z 506.423,A -85,B 0,C 180,E1 -26781.581,E2 -26781.581} C_VEL
LIN {X 0,Y 148.524,Z 495.877,A -85,B 0,C 180,E1 -26784.13,E2 -26784.13} C_VEL
LIN {X 0,Y 154.734,Z 485.156,A -85,B 0,C 180,E1 -26785.988,E2 -26785.988} C_VEL
LIN {X 0,Y 157.789,Z 479.033,A -85,B 0,C 180,E1 -26786.8,E2 -26786.8} C_VEL
LIN {X 0,Y 159.759,Z 473.917,A -85,B 0,C 180,E1 -26787.589,E2 -26787.589} C_VEL
LIN {X 0,Y 161.737,Z 465.431,A -85,B 0,C 180,E1 -26789.293,E2 -26789.293} C_VEL
LIN {X 0,Y 162.971,Z 458.497,A -85,B 0,C 180,E1 -26790.587,E2 -26790.587} C_VEL
LIN {X 0,Y 164.062,Z 453.029,A -85,B 0,C 180,E1 -26791.275,E2 -26791.275} C_VEL
LIN {X 0,Y 164.458,Z 451.15,A -85,B 0,C 180,E1 -26791.428,E2 -26791.428} C_VEL
LIN {X 0,Y 167.125,Z 437.796,A -85,B 0,C 180,E1 -26792.02,E2 -26792.02} C_VEL
LIN {X 0,Y 168.047,Z 429.505,A -85,B 0,C 180,E1 -26792.329,E2 -26792.329} C_VEL
LIN {X 0,Y 165.368,Z 421.263,A -85,B 0,C 180,E1 -26795.604,E2 -26795.604} C_VEL
LIN {X 0,Y 163.098,Z 415.068,A -85,B 0,C 180,E1 -26798.845,E2 -26798.845} C_VEL
LIN {X 0,Y 161.662,Z 411.426,A -85,B 0,C 180,E1 -26801.299,E2 -26801.299} C_VEL
LIN {X 0,Y 160.558,Z 409.218,A -85,B 0,C 180,E1 -26803.429,E2 -26803.429} C_VEL
LIN {X 0,Y 158.789,Z 405.507,A -85,B 0,C 180,E1 -26808.186,E2 -26808.186} C_VEL
LIN {X 0,Y 157.798,Z 404.254,A -85,B 0,C 180,E1 -26813.322,E2 -26813.322} C_VEL
LIN {X 0,Y 157.852,Z 403.98,A -85,B 0,C 180,E1 -26817.448,E2 -26817.448} C_VEL
LIN {X 0,Y 159.006,Z 405.639,A -85,B 0,C 180,E1 -26823.008,E2 -26823.008} C_VEL
LIN {X 0,Y 161.013,Z 409.889,A -85,B 0,C 180,E1 -26827.997,E2 -26827.997} C_VEL
LIN {X 0,Y 162.963,Z 413.799,A -85,B 0,C 180,E1 -26831.347,E2 -26831.347} C_VEL
LIN {X 0,Y 165.494,Z 418.792,A -85,B 0,C 180,E1 -26834.761,E2 -26834.761} C_VEL
LIN {X 0,Y 168.418,Z 425.171,A -85,B 0,C 180,E1 -26838.057,E2 -26838.057} C_VEL
LIN {X 0,Y 166.62,Z 438.425,A -85,B 0,C 180,E1 -26838.577,E2 -26838.577} C_VEL
LIN {X 0,Y 163.418,Z 451.907,A -85,B 0,C 180,E1 -26839.359,E2 -26839.359} C_VEL
LIN {X 0,Y 159.727,Z 463.143,A -85,B 0,C 180,E1 -26840.321,E2 -26840.321} C_VEL
LIN {X 0,Y 154.813,Z 474.85,A -85,B 0,C 180,E1 -26841.736,E2 -26841.736} C_VEL
LIN {X 0,Y 149.991,Z 484.026,A -85,B 0,C 180,E1 -26843.138,E2 -26843.138} C_VEL
LIN {X 0,Y 143.729,Z 494.08,A -85,B 0,C 180,E1 -26845.228,E2 -26845.228} C_VEL
LIN {X 0,Y 137.112,Z 502.91,A -85,B 0,C 180,E1 -26847.607,E2 -26847.607} C_VEL
LIN {X 0,Y 130.344,Z 510.617,A -85,B 0,C 180,E1 -26850.377,E2 -26850.377} C_VEL
LIN {X 0,Y 122.924,Z 517.915,A -85,B 0,C 180,E1 -26854,E2 -26854} C_VEL
LIN {X 0,Y 116.056,Z 523.688,A -85,B 0,C 180,E1 -26858.07,E2 -26858.07} C_VEL
LIN {X 0,Y 109.772,Z 528.193,A -85,B 0,C 180,E1 -26862.583,E2 -26862.583} C_VEL
LIN {X 0,Y 103.841,Z 531.821,A -85,B 0,C 180,E1 -26868.114,E2 -26868.114} C_VEL
LIN {X 0,Y 98.259,Z 534.492,A -85,B 0,C 180,E1 -26875.094,E2 -26875.094} C_VEL
LIN {X 0,Y 95.899,Z 535.329,A -85,B 0,C 180,E1 -26879.134,E2 -26879.134} C_VEL
LIN {X 0,Y 93.69,Z 535.74,A -85,B 0,C 180,E1 -26884.178,E2 -26884.178} C_VEL
LIN {X 0,Y 91.481,Z 535.31,A -85,B 0,C 180,E1 -26892.101,E2 -26892.101} C_VEL
LIN {X 0,Y 90.91,Z 534.509,A -85,B 0,C 180,E1 -26896.588,E2 -26896.588} C_VEL
LIN {X 0,Y 90.779,Z 533.263,A -85,B 0,C 180,E1 -26901.09,E2 -26901.09} C_VEL
LIN {X 0,Y 91.441,Z 530.712,A -85,B 0,C 180,E1 -26907.632,E2 -26907.632} C_VEL
LIN {X 0,Y 92.683,Z 527.021,A -85,B 0,C 180,E1 -26914.346,E2 -26914.346} C_VEL
LIN {X 0,Y 94.866,Z 522.304,A -85,B 0,C 180,E1 -26920.671,E2 -26920.671} C_VEL
LIN {X 0,Y 98.581,Z 515.226,A -85,B 0,C 180,E1 -26927.635,E2 -26927.635} C_VEL
LIN {X 0,Y 102.729,Z 507.54,A -85,B 0,C 180,E1 -26933.162,E2 -26933.162} C_VEL
LIN {X 0,Y 106.768,Z 499.677,A -85,B 0,C 180,E1 -26937.434,E2 -26937.434} C_VEL
LIN {X 0,Y 111.424,Z 490.066,A -85,B 0,C 180,E1 -26941.354,E2 -26941.354} C_VEL
LIN {X 0,Y 115.944,Z 479.403,A -85,B 0,C 180,E1 -26944.627,E2 -26944.627} C_VEL
LIN {X 0,Y 119.818,Z 469.05,A -85,B 0,C 180,E1 -26946.955,E2 -26946.955} C_VEL
LIN {X 0,Y 123.017,Z 457.86,A -85,B 0,C 180,E1 -26948.932,E2 -26948.932} C_VEL
LIN {X 0,Y 125.694,Z 444.737,A -85,B 0,C 180,E1 -26950.651,E2 -26950.651} C_VEL
LIN {X 0,Y 127.824,Z 431.394,A -85,B 0,C 180,E1 -26951.647,E2 -26951.647} C_VEL
LIN {X 0,Y 130.947,Z 393.326,A -85,B 0,C 180,E1 -26953.315,E2 -26953.315} C_VEL
LIN {X 0,Y 126.671,Z 383.959,A -85,B 0,C 180,E1 -26956.424,E2 -26956.424} C_VEL
LIN {X 0,Y 121.947,Z 375.444,A -85,B 0,C 180,E1 -26960.229,E2 -26960.229} C_VEL
LIN {X 0,Y 117.643,Z 368.605,A -85,B 0,C 180,E1 -26964.253,E2 -26964.253} C_VEL
LIN {X 0,Y 115.138,Z 364.897,A -85,B 0,C 180,E1 -26966.953,E2 -26966.953} C_VEL
LIN {X 0,Y 112.489,Z 361.023,A -85,B 0,C 180,E1 -26970.243,E2 -26970.243} C_VEL
LIN {X 0,Y 109.889,Z 357.66,A -85,B 0,C 180,E1 -26974.044,E2 -26974.044} C_VEL
LIN {X 0,Y 109.205,Z 356.372,A -85,B 0,C 180,E1 -26975.272,E2 -26975.272} C_VEL
LIN {X 0,Y 106.568,Z 353.834,A -85,B 0,C 180,E1 -26980.497,E2 -26980.497} C_VEL
LIN {X 0,Y 105.333,Z 350.927,A -85,B 0,C 180,E1 -26984.521,E2 -26984.521} C_VEL
LIN {X 0,Y 103.815,Z 350.043,A -85,B 0,C 180,E1 -26996.119,E2 -26996.119} C_VEL
LIN {X 0,Y 104.379,Z 350.162,A -85,B 0,C 180,E1 -27000.965,E2 -27000.965} C_VEL
LIN {X 0,Y 105.724,Z 351.135,A -85,B 0,C 180,E1 -27006.172,E2 -27006.172} C_VEL
LIN {X 0,Y 107.456,Z 354.618,A -85,B 0,C 180,E1 -27010.958,E2 -27010.958} C_VEL
LIN {X 0,Y 109.54,Z 356.709,A -85,B 0,C 180,E1 -27014.78,E2 -27014.78} C_VEL
LIN {X 0,Y 111.785,Z 360.219,A -85,B 0,C 180,E1 -27018.322,E2 -27018.322} C_VEL
LIN {X 0,Y 113.059,Z 361.704,A -85,B 0,C 180,E1 -27019.993,E2 -27019.993} C_VEL
LIN {X 0,Y 116.436,Z 366.664,A -85,B 0,C 180,E1 -27023.968,E2 -27023.968} C_VEL
LIN {X 0,Y 119.63,Z 371.586,A -85,B 0,C 180,E1 -27027.173,E2 -27027.173} C_VEL
LIN {X 0,Y 123.485,Z 378.106,A -85,B 0,C 180,E1 -27030.566,E2 -27030.566} C_VEL
LIN {X 0,Y 125.486,Z 382.358,A -85,B 0,C 180,E1 -27032.225,E2 -27032.225} C_VEL
LIN {X 0,Y 128.65,Z 391.155,A -85,B 0,C 180,E1 -27034.807,E2 -27034.807} C_VEL
LIN {X 0,Y 130.406,Z 397.169,A -85,B 0,C 180,E1 -27036.224,E2 -27036.224} C_VEL
LIN {X 0,Y 130.375,Z 402.592,A -85,B 0,C 180,E1 -27036.654,E2 -27036.654} C_VEL
LIN {X 0,Y 127.361,Z 438.943,A -85,B 0,C 180,E1 -27038.288,E2 -27038.288} C_VEL
LIN {X 0,Y 125.2,Z 452.199,A -85,B 0,C 180,E1 -27039.326,E2 -27039.326} C_VEL
LIN {X 0,Y 122.377,Z 464.265,A -85,B 0,C 180,E1 -27040.773,E2 -27040.773} C_VEL
LIN {X 0,Y 118.551,Z 476.413,A -85,B 0,C 180,E1 -27042.813,E2 -27042.813} C_VEL
LIN {X 0,Y 114.085,Z 487.982,A -85,B 0,C 180,E1 -27045.517,E2 -27045.517} C_VEL
LIN {X 0,Y 110.004,Z 497.341,A -85,B 0,C 180,E1 -27048.486,E2 -27048.486} C_VEL
LIN {X 0,Y 105.87,Z 506.057,A -85,B 0,C 180,E1 -27052.12,E2 -27052.12} C_VEL
LIN {X 0,Y 101.536,Z 514.044,A -85,B 0,C 180,E1 -27056.38,E2 -27056.38} C_VEL
LIN {X 0,Y 98.873,Z 519.452,A -85,B 0,C 180,E1 -27060.164,E2 -27060.164} C_VEL
LIN {X 0,Y 95.36,Z 526.206,A -85,B 0,C 180,E1 -27066.09,E2 -27066.09} C_VEL
LIN {X 0,Y 92.863,Z 531.584,A -85,B 0,C 180,E1 -27072.381,E2 -27072.381} C_VEL
LIN {X 0,Y 91.503,Z 535.766,A -85,B 0,C 180,E1 -27078.932,E2 -27078.932} C_VEL
LIN {X 0,Y 91.013,Z 538.855,A -85,B 0,C 180,E1 -27085.574,E2 -27085.574} C_VEL
LIN {X 0,Y 91.162,Z 540.379,A -85,B 0,C 180,E1 -27090.002,E2 -27090.002} C_VEL
LIN {X 0,Y 91.003,Z 541.411,A -85,B 0,C 180,E1 -27094.432,E2 -27094.432} C_VEL
LIN {X 0,Y 91.913,Z 542.3,A -85,B 0,C 180,E1 -27103.263,E2 -27103.263} C_VEL
LIN {X 0,Y 93.036,Z 542.174,A -85,B 0,C 180,E1 -27107.59,E2 -27107.59} C_VEL
LIN {X 0,Y 94.635,Z 541.638,A -85,B 0,C 180,E1 -27111.799,E2 -27111.799} C_VEL
LIN {X 0,Y 99.469,Z 539.385,A -85,B 0,C 180,E1 -27119.645,E2 -27119.645} C_VEL
LIN {X 0,Y 104.227,Z 536.626,A -85,B 0,C 180,E1 -27124.972,E2 -27124.972} C_VEL
LIN {X 0,Y 109.722,Z 532.871,A -85,B 0,C 180,E1 -27129.833,E2 -27129.833} C_VEL
LIN {X 0,Y 115.956,Z 528.025,A -85,B 0,C 180,E1 -27134.189,E2 -27134.189} C_VEL
LIN {X 0,Y 122.922,Z 521.94,A -85,B 0,C 180,E1 -27138.012,E2 -27138.012} C_VEL
LIN {X 0,Y 130.422,Z 514.398,A -85,B 0,C 180,E1 -27141.387,E2 -27141.387} C_VEL
LIN {X 0,Y 136.997,Z 506.715,A -85,B 0,C 180,E1 -27143.901,E2 -27143.901} C_VEL
LIN {X 0,Y 144.494,Z 496.316,A -85,B 0,C 180,E1 -27146.403,E2 -27146.403} C_VEL
LIN {X 0,Y 150.887,Z 485.743,A -85,B 0,C 180,E1 -27148.218,E2 -27148.218} C_VEL
LIN {X 0,Y 156.775,Z 473.893,A -85,B 0,C 180,E1 -27149.651,E2 -27149.651} C_VEL
LIN {X 0,Y 161.632,Z 461.076,A -85,B 0,C 180,E1 -27150.776,E2 -27150.776} C_VEL
LIN {X 0,Y 164.458,Z 451.15,A -85,B 0,C 180,E1 -27151.428,E2 -27151.428} C_VEL
LIN {X 0,Y 165.377,Z 445.552,A -85,B 0,C 180,E1 -27151.996,E2 -27151.996} C_VEL
LIN {X 0,Y 165.517,Z 440.241,A -85,B 0,C 180,E1 -27152.911,E2 -27152.911} C_VEL
LIN {X 0,Y 165.09,Z 435.322,A -85,B 0,C 180,E1 -27154.087,E2 -27154.087} C_VEL
LIN {X 0,Y 164.259,Z 430.812,A -85,B 0,C 180,E1 -27155.474,E2 -27155.474} C_VEL
LIN {X 0,Y 162.859,Z 425.557,A -85,B 0,C 180,E1 -27157.582,E2 -27157.582} C_VEL
LIN {X 0,Y 161.237,Z 420.747,A -85,B 0,C 180,E1 -27160.256,E2 -27160.256} C_VEL
LIN {X 0,Y 160.188,Z 417.794,A -85,B 0,C 180,E1 -27162.279,E2 -27162.279} C_VEL
LIN {X 0,Y 159.223,Z 415.823,A -85,B 0,C 180,E1 -27164.314,E2 -27164.314} C_VEL
LIN {X 0,Y 157.784,Z 412.466,A -85,B 0,C 180,E1 -27168.598,E2 -27168.598} C_VEL
LIN {X 0,Y 156.928,Z 411.319,A -85,B 0,C 180,E1 -27173.285,E2 -27173.285} C_VEL
LIN {X 0,Y 157.047,Z 411.124,A -85,B 0,C 180,E1 -27178.076,E2 -27178.076} C_VEL
LIN {X 0,Y 157.968,Z 412.61,A -85,B 0,C 180,E1 -27182.55,E2 -27182.55} C_VEL
LIN {X 0,Y 159.862,Z 416.909,A -85,B 0,C 180,E1 -27187.578,E2 -27187.578} C_VEL
LIN {X 0,Y 161.542,Z 420.539,A -85,B 0,C 180,E1 -27190.655,E2 -27190.655} C_VEL
LIN {X 0,Y 163.823,Z 425.395,A -85,B 0,C 180,E1 -27193.964,E2 -27193.964} C_VEL
LIN {X 0,Y 165.336,Z 429.183,A -85,B 0,C 180,E1 -27195.943,E2 -27195.943} C_VEL
LIN {X 0,Y 163.081,Z 442.566,A -85,B 0,C 180,E1 -27196.491,E2 -27196.491} C_VEL
LIN {X 0,Y 159.871,Z 454.569,A -85,B 0,C 180,E1 -27197.217,E2 -27197.217} C_VEL
LIN {X 0,Y 156.144,Z 465.112,A -85,B 0,C 180,E1 -27198.158,E2 -27198.158} C_VEL
LIN {X 0,Y 150.737,Z 477.035,A -85,B 0,C 180,E1 -27199.612,E2 -27199.612} C_VEL
LIN {X 0,Y 145.824,Z 485.797,A -85,B 0,C 180,E1 -27200.967,E2 -27200.967} C_VEL
LIN {X 0,Y 139.35,Z 495.591,A -85,B 0,C 180,E1 -27203.01,E2 -27203.01} C_VEL
LIN {X 0,Y 132.306,Z 504.465,A -85,B 0,C 180,E1 -27205.439,E2 -27205.439} C_VEL
LIN {X 0,Y 124.167,Z 513.026,A -85,B 0,C 180,E1 -27208.677,E2 -27208.677} C_VEL
LIN {X 0,Y 116.504,Z 519.858,A -85,B 0,C 180,E1 -27212.375,E2 -27212.375} C_VEL
LIN {X 0,Y 109.399,Z 525.279,A -85,B 0,C 180,E1 -27216.578,E2 -27216.578} C_VEL
LIN {X 0,Y 102.907,Z 529.476,A -85,B 0,C 180,E1 -27221.3,E2 -27221.3} C_VEL
LIN {X 0,Y 97.982,Z 532.19,A -85,B 0,C 180,E1 -27225.829,E2 -27225.829} C_VEL
LIN {X 0,Y 92.372,Z 534.656,A -85,B 0,C 180,E1 -27232.504,E2 -27232.504} C_VEL
LIN {X 0,Y 89.711,Z 535.532,A -85,B 0,C 180,E1 -27236.741,E2 -27236.741} C_VEL
LIN {X 0,Y 86.954,Z 536.013,A -85,B 0,C 180,E1 -27242.756,E2 -27242.756} C_VEL
LIN {X 0,Y 84.614,Z 535.626,A -85,B 0,C 180,E1 -27250.593,E2 -27250.593} C_VEL
LIN {X 0,Y 83.912,Z 534.867,A -85,B 0,C 180,E1 -27255.445,E2 -27255.445} C_VEL
LIN {X 0,Y 83.665,Z 533.668,A -85,B 0,C 180,E1 -27260.326,E2 -27260.326} C_VEL
LIN {X 0,Y 84.385,Z 530.905,A -85,B 0,C 180,E1 -27268.035,E2 -27268.035} C_VEL
LIN {X 0,Y 85.61,Z 527.549,A -85,B 0,C 180,E1 -27274.706,E2 -27274.706} C_VEL
LIN {X 0,Y 87.892,Z 522.904,A -85,B 0,C 180,E1 -27281.529,E2 -27281.529} C_VEL
LIN {X 0,Y 91.865,Z 515.902,A -85,B 0,C 180,E1 -27288.971,E2 -27288.971} C_VEL
LIN {X 0,Y 96.24,Z 508.335,A -85,B 0,C 180,E1 -27294.825,E2 -27294.825} C_VEL
LIN {X 0,Y 100.532,Z 500.593,A -85,B 0,C 180,E1 -27299.295,E2 -27299.295} C_VEL
LIN {X 0,Y 105.964,Z 490.052,A -85,B 0,C 180,E1 -27303.74,E2 -27303.74} C_VEL
LIN {X 0,Y 110.749,Z 479.332,A -85,B 0,C 180,E1 -27307.072,E2 -27307.072} C_VEL
LIN {X 0,Y 114.822,Z 468.889,A -85,B 0,C 180,E1 -27309.419,E2 -27309.419} C_VEL
LIN {X 0,Y 118.177,Z 457.55,A -85,B 0,C 180,E1 -27311.419,E2 -27311.419} C_VEL
LIN {X 0,Y 121.032,Z 444.121,A -85,B 0,C 180,E1 -27313.162,E2 -27313.162} C_VEL
LIN {X 0,Y 123.157,Z 431.126,A -85,B 0,C 180,E1 -27314.085,E2 -27314.085} C_VEL
LIN {X 0,Y 126.188,Z 395.844,A -85,B 0,C 180,E1 -27315.629,E2 -27315.629} C_VEL
LIN {X 0,Y 122.504,Z 387.647,A -85,B 0,C 180,E1 -27318.624,E2 -27318.624} C_VEL
LIN {X 0,Y 117.675,Z 378.699,A -85,B 0,C 180,E1 -27323.041,E2 -27323.041} C_VEL
LIN {X 0,Y 113.307,Z 371.583,A -85,B 0,C 180,E1 -27327.837,E2 -27327.837} C_VEL
LIN {X 0,Y 110.536,Z 367.404,A -85,B 0,C 180,E1 -27331.52,E2 -27331.52} C_VEL
LIN {X 0,Y 108.081,Z 363.95,A -85,B 0,C 180,E1 -27335.47,E2 -27335.47} C_VEL
LIN {X 0,Y 107.341,Z 362.884,A -85,B 0,C 180,E1 -27336.869,E2 -27336.869} C_VEL
LIN {X 0,Y 104.863,Z 359.843,A -85,B 0,C 180,E1 -27342.699,E2 -27342.699} C_VEL
LIN {X 0,Y 104.199,Z 357.901,A -85,B 0,C 180,E1 -27345.35,E2 -27345.35} C_VEL
LIN {X 0,Y 102.943,Z 357.092,A -85,B 0,C 180,E1 -27356.086,E2 -27356.086} C_VEL
LIN {X 0,Y 103.46,Z 357.19,A -85,B 0,C 180,E1 -27360.73,E2 -27360.73} C_VEL
LIN {X 0,Y 104.524,Z 358.025,A -85,B 0,C 180,E1 -27365.228,E2 -27365.228} C_VEL
LIN {X 0,Y 106.304,Z 361.643,A -85,B 0,C 180,E1 -27370.488,E2 -27370.488} C_VEL
LIN {X 0,Y 107.883,Z 363.316,A -85,B 0,C 180,E1 -27373.592,E2 -27373.592} C_VEL
LIN {X 0,Y 110.102,Z 366.854,A -85,B 0,C 180,E1 -27377.351,E2 -27377.351} C_VEL
LIN {X 0,Y 111.112,Z 368.213,A -85,B 0,C 180,E1 -27378.796,E2 -27378.796} C_VEL
LIN {X 0,Y 114.209,Z 373.003,A -85,B 0,C 180,E1 -27382.739,E2 -27382.739} C_VEL
LIN {X 0,Y 117.875,Z 378.945,A -85,B 0,C 180,E1 -27386.643,E2 -27386.643} C_VEL
LIN {X 0,Y 121.329,Z 385.589,A -85,B 0,C 180,E1 -27389.886,E2 -27389.886} C_VEL
LIN {X 0,Y 124.534,Z 394.908,A -85,B 0,C 180,E1 -27392.824,E2 -27392.824} C_VEL
LIN {X 0,Y 125.823,Z 399.941,A -85,B 0,C 180,E1 -27394.028,E2 -27394.028} C_VEL
LIN {X 0,Y 125.367,Z 407.812,A -85,B 0,C 180,E1 -27394.475,E2 -27394.475} C_VEL
LIN {X 0,Y 122.547,Z 439.297,A -85,B 0,C 180,E1 -27395.901,E2 -27395.901} C_VEL
LIN {X 0,Y 120.161,Z 452.973,A -85,B 0,C 180,E1 -27396.995,E2 -27396.995} C_VEL
LIN {X 0,Y 116.879,Z 465.753,A -85,B 0,C 180,E1 -27398.588,E2 -27398.588} C_VEL
LIN {X 0,Y 112.598,Z 478.278,A -85,B 0,C 180,E1 -27400.821,E2 -27400.821} C_VEL
LIN {X 0,Y 108.536,Z 488.16,A -85,B 0,C 180,E1 -27403.246,E2 -27403.246} C_VEL
LIN {X 0,Y 104.236,Z 497.444,A -85,B 0,C 180,E1 -27406.287,E2 -27406.287} C_VEL
LIN {X 0,Y 99.381,Z 506.975,A -85,B 0,C 180,E1 -27410.475,E2 -27410.475} C_VEL
LIN {X 0,Y 95.137,Z 514.212,A -85,B 0,C 180,E1 -27414.59,E2 -27414.59} C_VEL
LIN {X 0,Y 92.76,Z 518.779,A -85,B 0,C 180,E1 -27417.974,E2 -27417.974} C_VEL
LIN {X 0,Y 88.893,Z 525.606,A -85,B 0,C 180,E1 -27424.228,E2 -27424.228} C_VEL
LIN {X 0,Y 86.076,Z 531.049,A -85,B 0,C 180,E1 -27430.941,E2 -27430.941} C_VEL
LIN {X 0,Y 84.508,Z 535.294,A -85,B 0,C 180,E1 -27438.003,E2 -27438.003} C_VEL
LIN {X 0,Y 83.922,Z 538.442,A -85,B 0,C 180,E1 -27445.199,E2 -27445.199} C_VEL
LIN {X 0,Y 84.08,Z 540,A -85,B 0,C 180,E1 -27450.003,E2 -27450.003} C_VEL
LIN {X 0,Y 83.914,Z 541.08,A -85,B 0,C 180,E1 -27454.807,E2 -27454.807} C_VEL
LIN {X 0,Y 84.994,Z 542.021,A -85,B 0,C 180,E1 -27464.365,E2 -27464.365} C_VEL
LIN {X 0,Y 88.05,Z 541.435,A -85,B 0,C 180,E1 -27473.524,E2 -27473.524} C_VEL
LIN {X 0,Y 93.332,Z 539.239,A -85,B 0,C 180,E1 -27481.813,E2 -27481.813} C_VEL
LIN {X 0,Y 98.486,Z 536.537,A -85,B 0,C 180,E1 -27487.344,E2 -27487.344} C_VEL
LIN {X 0,Y 104.367,Z 532.841,A -85,B 0,C 180,E1 -27492.332,E2 -27492.332} C_VEL
LIN {X 0,Y 110.96,Z 528.058,A -85,B 0,C 180,E1 -27496.753,E2 -27496.753} C_VEL
LIN {X 0,Y 118.293,Z 522.043,A -85,B 0,C 180,E1 -27500.568,E2 -27500.568} C_VEL
LIN {X 0,Y 126.108,Z 514.58,A -85,B 0,C 180,E1 -27503.911,E2 -27503.911} C_VEL
LIN {X 0,Y 132.95,Z 506.987,A -85,B 0,C 180,E1 -27506.366,E2 -27506.366} C_VEL
LIN {X 0,Y 139.97,Z 497.812,A -85,B 0,C 180,E1 -27508.605,E2 -27508.605} C_VEL
LIN {X 0,Y 146.554,Z 487.614,A -85,B 0,C 180,E1 -27510.365,E2 -27510.365} C_VEL
LIN {X 0,Y 152.561,Z 476.317,A -85,B 0,C 180,E1 -27511.768,E2 -27511.768} C_VEL
LIN {X 0,Y 157.501,Z 464.606,A -85,B 0,C 180,E1 -27512.831,E2 -27512.831} C_VEL
LIN {X 0,Y 161.506,Z 451.719,A -85,B 0,C 180,E1 -27513.684,E2 -27513.684} C_VEL
LIN {X 0,Y 164.123,Z 439.347,A -85,B 0,C 180,E1 -27514.246,E2 -27514.246} C_VEL
LIN {X 0,Y 165.017,Z 432.654,A -85,B 0,C 180,E1 -27514.507,E2 -27514.507} C_VEL
LIN {X 0,Y 162.859,Z 425.557,A -85,B 0,C 180,E1 -27517.582,E2 -27517.582} C_VEL
LIN {X 0,Y 162.014,Z 423.871,A -85,B 0,C 180,E1 -27518.787,E2 -27518.787} C_VEL
LIN {X 0,Y 160.689,Z 423.101,A -85,B 0,C 180,E1 -27520.586,E2 -27520.586} C_VEL
LIN {X 0,Y 158.269,Z 422.871,A -85,B 0,C 180,E1 -27524.439,E2 -27524.439} C_VEL
LIN {X 0,Y 158.047,Z 422.633,A -85,B 0,C 180,E1 -27524.923,E2 -27524.923} C_VEL
LIN {X 0,Y 156.702,Z 419.339,A -85,B 0,C 180,E1 -27529.336,E2 -27529.336} C_VEL
LIN {X 0,Y 155.977,Z 418.233,A -85,B 0,C 180,E1 -27534.829,E2 -27534.829} C_VEL
LIN {X 0,Y 156.233,Z 418.275,A -85,B 0,C 180,E1 -27538.55,E2 -27538.55} C_VEL
LIN {X 0,Y 156.94,Z 419.588,A -85,B 0,C 180,E1 -27542.085,E2 -27542.085} C_VEL
LIN {X 0,Y 158.512,Z 423.428,A -85,B 0,C 180,E1 -27546.683,E2 -27546.683} C_VEL
LIN {X 0,Y 160.021,Z 426.926,A -85,B 0,C 180,E1 -27549.719,E2 -27549.719} C_VEL
LIN {X 0,Y 162.057,Z 431.935,A -85,B 0,C 180,E1 -27553.128,E2 -27553.128} C_VEL
LIN {X 0,Y 162.42,Z 432.843,A -85,B 0,C 180,E1 -27553.68,E2 -27553.68} C_VEL
LIN {X 0,Y 159.794,Z 446.081,A -85,B 0,C 180,E1 -27554.309,E2 -27554.309} C_VEL
LIN {X 0,Y 156.152,Z 458.148,A -85,B 0,C 180,E1 -27555.062,E2 -27555.062} C_VEL
LIN {X 0,Y 151.459,Z 470.073,A -85,B 0,C 180,E1 -27556.234,E2 -27556.234} C_VEL
LIN {X 0,Y 145.637,Z 481.305,A -85,B 0,C 180,E1 -27557.62,E2 -27557.62} C_VEL
LIN {X 0,Y 138.901,Z 492.038,A -85,B 0,C 180,E1 -27559.544,E2 -27559.544} C_VEL
LIN {X 0,Y 132.397,Z 500.6,A -85,B 0,C 180,E1 -27561.551,E2 -27561.551} C_VEL
LIN {X 0,Y 125.062,Z 508.738,A -85,B 0,C 180,E1 -27564.048,E2 -27564.048} C_VEL
LIN {X 0,Y 116.752,Z 516.479,A -85,B 0,C 180,E1 -27567.389,E2 -27567.389} C_VEL
LIN {X 0,Y 107.665,Z 523.571,A -85,B 0,C 180,E1 -27571.938,E2 -27571.938} C_VEL
LIN {X 0,Y 100.484,Z 528.238,A -85,B 0,C 180,E1 -27576.452,E2 -27576.452} C_VEL
LIN {X 0,Y 94.019,Z 531.757,A -85,B 0,C 180,E1 -27581.622,E2 -27581.622} C_VEL
LIN {X 0,Y 90.164,Z 533.508,A -85,B 0,C 180,E1 -27585.448,E2 -27585.448} C_VEL
LIN {X 0,Y 86.702,Z 534.82,A -85,B 0,C 180,E1 -27589.571,E2 -27589.571} C_VEL
LIN {X 0,Y 83.724,Z 535.727,A -85,B 0,C 180,E1 -27594.011,E2 -27594.011} C_VEL
LIN {X 0,Y 80.268,Z 536.287,A -85,B 0,C 180,E1 -27601.111,E2 -27601.111} C_VEL
LIN {X 0,Y 77.826,Z 535.941,A -85,B 0,C 180,E1 -27608.823,E2 -27608.823} C_VEL
LIN {X 0,Y 76.927,Z 535.214,A -85,B 0,C 180,E1 -27614.09,E2 -27614.09} C_VEL
LIN {X 0,Y 76.584,Z 534.072,A -85,B 0,C 180,E1 -27619.421,E2 -27619.421} C_VEL
LIN {X 0,Y 77.332,Z 531.078,A -85,B 0,C 180,E1 -27628.561,E2 -27628.561} C_VEL
LIN {X 0,Y 79.165,Z 526.652,A -85,B 0,C 180,E1 -27637.65,E2 -27637.65} C_VEL
LIN {X 0,Y 82.045,Z 521.688,A -85,B 0,C 180,E1 -27644.888,E2 -27644.888} C_VEL
LIN {X 0,Y 85.896,Z 515.464,A -85,B 0,C 180,E1 -27651.601,E2 -27651.601} C_VEL
LIN {X 0,Y 90.704,Z 507.689,A -85,B 0,C 180,E1 -27657.701,E2 -27657.701} C_VEL
LIN {X 0,Y 96.434,Z 497.962,A -85,B 0,C 180,E1 -27663.13,E2 -27663.13} C_VEL
LIN {X 0,Y 101.802,Z 487.869,A -85,B 0,C 180,E1 -27667.158,E2 -27667.158} C_VEL
LIN {X 0,Y 107.005,Z 476.426,A -85,B 0,C 180,E1 -27670.431,E2 -27670.431} C_VEL
LIN {X 0,Y 111.256,Z 465.191,A -85,B 0,C 180,E1 -27672.768,E2 -27672.768} C_VEL
LIN {X 0,Y 114.756,Z 452.627,A -85,B 0,C 180,E1 -27674.769,E2 -27674.769} C_VEL
LIN {X 0,Y 116.964,Z 441.91,A -85,B 0,C 180,E1 -27675.982,E2 -27675.982} C_VEL
LIN {X 0,Y 118.917,Z 429.033,A -85,B 0,C 180,E1 -27676.799,E2 -27676.799} C_VEL
LIN {X 0,Y 121.633,Z 398.408,A -85,B 0,C 180,E1 -27678.125,E2 -27678.125} C_VEL
LIN {X 0,Y 118.139,Z 390.597,A -85,B 0,C 180,E1 -27681.345,E2 -27681.345} C_VEL
LIN {X 0,Y 114.661,Z 383.955,A -85,B 0,C 180,E1 -27684.936,E2 -27684.936} C_VEL
LIN {X 0,Y 111.059,Z 377.683,A -85,B 0,C 180,E1 -27689.315,E2 -27689.315} C_VEL
LIN {X 0,Y 108.508,Z 373.661,A -85,B 0,C 180,E1 -27693.039,E2 -27693.039} C_VEL
LIN {X 0,Y 105.915,Z 369.656,A -85,B 0,C 180,E1 -27697.815,E2 -27697.815} C_VEL
LIN {X 0,Y 103.501,Z 366.254,A -85,B 0,C 180,E1 -27704.24,E2 -27704.24} C_VEL
LIN {X 0,Y 103.089,Z 364.864,A -85,B 0,C 180,E1 -27706.196,E2 -27706.196} C_VEL
LIN {X 0,Y 102.071,Z 364.14,A -85,B 0,C 180,E1 -27716.052,E2 -27716.052} C_VEL
LIN {X 0,Y 102.712,Z 364.383,A -85,B 0,C 180,E1 -27721.471,E2 -27721.471} C_VEL
LIN {X 0,Y 103.383,Z 364.98,A -85,B 0,C 180,E1 -27724.387,E2 -27724.387} C_VEL
LIN {X 0,Y 105.204,Z 368.697,A -85,B 0,C 180,E1 -27730.106,E2 -27730.106} C_VEL
LIN {X 0,Y 106.332,Z 370.061,A -85,B 0,C 180,E1 -27732.497,E2 -27732.497} C_VEL
LIN {X 0,Y 108.665,Z 373.744,A -85,B 0,C 180,E1 -27736.679,E2 -27736.679} C_VEL
LIN {X 0,Y 111.905,Z 379.084,A -85,B 0,C 180,E1 -27741.29,E2 -27741.29} C_VEL
LIN {X 0,Y 115.124,Z 384.694,A -85,B 0,C 180,E1 -27745.057,E2 -27745.057} C_VEL
LIN {X 0,Y 117.945,Z 390.406,A -85,B 0,C 180,E1 -27747.986,E2 -27747.986} C_VEL
LIN {X 0,Y 120.629,Z 398.951,A -85,B 0,C 180,E1 -27750.772,E2 -27750.772} C_VEL
LIN {X 0,Y 121.444,Z 401.908,A -85,B 0,C 180,E1 -27751.593,E2 -27751.593} C_VEL
LIN {X 0,Y 118.164,Z 438.222,A -85,B 0,C 180,E1 -27753.231,E2 -27753.231} C_VEL
LIN {X 0,Y 115.842,Z 451.449,A -85,B 0,C 180,E1 -27754.252,E2 -27754.252} C_VEL
LIN {X 0,Y 112.591,Z 464.138,A -85,B 0,C 180,E1 -27755.765,E2 -27755.765} C_VEL
LIN {X 0,Y 108.75,Z 475.382,A -85,B 0,C 180,E1 -27757.664,E2 -27757.664} C_VEL
LIN {X 0,Y 105.05,Z 484.43,A -85,B 0,C 180,E1 -27759.707,E2 -27759.707} C_VEL
LIN {X 0,Y 100.248,Z 494.29,A -85,B 0,C 180,E1 -27762.603,E2 -27762.603} C_VEL
LIN {X 0,Y 94.962,Z 504.334,A -85,B 0,C 180,E1 -27766.801,E2 -27766.801} C_VEL
LIN {X 0,Y 90.031,Z 512.529,A -85,B 0,C 180,E1 -27771.359,E2 -27771.359} C_VEL
LIN {X 0,Y 85.971,Z 519.347,A -85,B 0,C 180,E1 -27776.513,E2 -27776.513} C_VEL
LIN {X 0,Y 82.524,Z 525.006,A -85,B 0,C 180,E1 -27782.073,E2 -27782.073} C_VEL
LIN {X 0,Y 79.338,Z 530.513,A -85,B 0,C 180,E1 -27789.251,E2 -27789.251} C_VEL
LIN {X 0,Y 77.555,Z 534.823,A -85,B 0,C 180,E1 -27796.909,E2 -27796.909} C_VEL
LIN {X 0,Y 76.855,Z 538.03,A -85,B 0,C 180,E1 -27804.756,E2 -27804.756} C_VEL
LIN {X 0,Y 76.985,Z 539.616,A -85,B 0,C 180,E1 -27810.003,E2 -27810.003} C_VEL
LIN {X 0,Y 76.849,Z 540.745,A -85,B 0,C 180,E1 -27815.25,E2 -27815.25} C_VEL
LIN {X 0,Y 78.122,Z 541.742,A -85,B 0,C 180,E1 -27825.66,E2 -27825.66} C_VEL
LIN {X 0,Y 81.56,Z 541.22,A -85,B 0,C 180,E1 -27835.524,E2 -27835.524} C_VEL
LIN {X 0,Y 84.226,Z 540.359,A -85,B 0,C 180,E1 -27840.046,E2 -27840.046} C_VEL
LIN {X 0,Y 90.956,Z 537.435,A -85,B 0,C 180,E1 -27848.183,E2 -27848.183} C_VEL
LIN {X 0,Y 97.597,Z 533.792,A -85,B 0,C 180,E1 -27853.936,E2 -27853.936} C_VEL
LIN {X 0,Y 103.8,Z 529.784,A -85,B 0,C 180,E1 -27858.142,E2 -27858.142} C_VEL
LIN {X 0,Y 111.273,Z 524.275,A -85,B 0,C 180,E1 -27862.141,E2 -27862.141} C_VEL
LIN {X 0,Y 119.301,Z 517.419,A -85,B 0,C 180,E1 -27865.564,E2 -27865.564} C_VEL
LIN {X 0,Y 127.723,Z 508.884,A -85,B 0,C 180,E1 -27868.529,E2 -27868.529} C_VEL
LIN {X 0,Y 134.968,Z 500.143,A -85,B 0,C 180,E1 -27870.717,E2 -27870.717} C_VEL
LIN {X 0,Y 142.443,Z 489.4,A -85,B 0,C 180,E1 -27872.638,E2 -27872.638} C_VEL
LIN {X 0,Y 148.576,Z 478.668,A -85,B 0,C 180,E1 -27873.995,E2 -27873.995} C_VEL
LIN {X 0,Y 154.015,Z 466.64,A -85,B 0,C 180,E1 -27875.087,E2 -27875.087} C_VEL
LIN {X 0,Y 158.329,Z 453.96,A -85,B 0,C 180,E1 -27875.941,E2 -27875.941} C_VEL
LIN {X 0,Y 161.404,Z 440.878,A -85,B 0,C 180,E1 -27876.529,E2 -27876.529} C_VEL
LIN {X 0,Y 162.195,Z 436.045,A -85,B 0,C 180,E1 -27876.71,E2 -27876.71} C_VEL
LIN {X 0,Y 160.406,Z 429.374,A -85,B 0,C 180,E1 -27879.899,E2 -27879.899} C_VEL
LIN {X 0,Y 158.83,Z 424.364,A -85,B 0,C 180,E1 -27883.119,E2 -27883.119} C_VEL
LIN {X 0,Y 158.047,Z 422.633,A -85,B 0,C 180,E1 -27884.923,E2 -27884.923} C_VEL
LIN {X 0,Y 157.154,Z 422.07,A -85,B 0,C 180,E1 -27887.043,E2 -27887.043} C_VEL
LIN {X 0,Y 155.897,Z 423.145,A -85,B 0,C 180,E1 -27890.632,E2 -27890.632} C_VEL
LIN {X 0,Y 155.135,Z 425.031,A -85,B 0,C 180,E1 -27895.024,E2 -27895.024} C_VEL
LIN {X 0,Y 155.152,Z 425.177,A -85,B 0,C 180,E1 -27896.507,E2 -27896.507} C_VEL
LIN {X 0,Y 155.42,Z 425.506,A -85,B 0,C 180,E1 -27899.028,E2 -27899.028} C_VEL
LIN {X 0,Y 155.925,Z 426.535,A -85,B 0,C 180,E1 -27901.614,E2 -27901.614} C_VEL
LIN {X 0,Y 157.272,Z 430.283,A -85,B 0,C 180,E1 -27906.092,E2 -27906.092} C_VEL
LIN {X 0,Y 158.668,Z 434.117,A -85,B 0,C 180,E1 -27909.4,E2 -27909.4} C_VEL
LIN {X 0,Y 159.615,Z 436.978,A -85,B 0,C 180,E1 -27911.429,E2 -27911.429} C_VEL
LIN {X 0,Y 156.714,Z 449.622,A -85,B 0,C 180,E1 -27912.056,E2 -27912.056} C_VEL
LIN {X 0,Y 152.419,Z 462.208,A -85,B 0,C 180,E1 -27912.88,E2 -27912.88} C_VEL
LIN {X 0,Y 147.075,Z 474.282,A -85,B 0,C 180,E1 -27914.122,E2 -27914.122} C_VEL
LIN {X 0,Y 141.278,Z 484.543,A -85,B 0,C 180,E1 -27915.456,E2 -27915.456} C_VEL
LIN {X 0,Y 134.341,Z 494.649,A -85,B 0,C 180,E1 -27917.301,E2 -27917.301} C_VEL
LIN {X 0,Y 126.76,Z 503.771,A -85,B 0,C 180,E1 -27919.515,E2 -27919.515} C_VEL
LIN {X 0,Y 117.876,Z 512.621,A -85,B 0,C 180,E1 -27922.459,E2 -27922.459} C_VEL
LIN {X 0,Y 109.402,Z 519.633,A -85,B 0,C 180,E1 -27925.923,E2 -27925.923} C_VEL
LIN {X 0,Y 101.383,Z 525.207,A -85,B 0,C 180,E1 -27929.941,E2 -27929.941} C_VEL
LIN {X 0,Y 93.91,Z 529.545,A -85,B 0,C 180,E1 -27934.59,E2 -27934.59} C_VEL
LIN {X 0,Y 86.804,Z 532.935,A -85,B 0,C 180,E1 -27940.369,E2 -27940.369} C_VEL
LIN {X 0,Y 81.298,Z 534.984,A -85,B 0,C 180,E1 -27946.242,E2 -27946.242} C_VEL
LIN {X 0,Y 75.109,Z 536.462,A -85,B 0,C 180,E1 -27955.843,E2 -27955.843} C_VEL
LIN {X 0,Y 72.872,Z 536.562,A -85,B 0,C 180,E1 -27961.167,E2 -27961.167} C_VEL
LIN {X 0,Y 71.136,Z 536.255,A -85,B 0,C 180,E1 -27966.72,E2 -27966.72} C_VEL
LIN {X 0,Y 69.995,Z 535.559,A -85,B 0,C 180,E1 -27972.466,E2 -27972.466} C_VEL
LIN {X 0,Y 69.506,Z 534.467,A -85,B 0,C 180,E1 -27978.33,E2 -27978.33} C_VEL
LIN {X 0,Y 70.287,Z 531.263,A -85,B 0,C 180,E1 -27989.158,E2 -27989.158} C_VEL
LIN {X 0,Y 72.144,Z 527.18,A -85,B 0,C 180,E1 -27998.399,E2 -27998.399} C_VEL
LIN {X 0,Y 75.187,Z 522.29,A -85,B 0,C 180,E1 -28006.282,E2 -28006.282} C_VEL
LIN {X 0,Y 79.366,Z 516.14,A -85,B 0,C 180,E1 -28013.48,E2 -28013.48} C_VEL
LIN {X 0,Y 84.493,Z 508.501,A -85,B 0,C 180,E1 -28019.935,E2 -28019.935} C_VEL
LIN {X 0,Y 90.577,Z 498.887,A -85,B 0,C 180,E1 -28025.583,E2 -28025.583} C_VEL
LIN {X 0,Y 96.269,Z 488.956,A -85,B 0,C 180,E1 -28029.698,E2 -28029.698} C_VEL
LIN {X 0,Y 101.703,Z 477.75,A -85,B 0,C 180,E1 -28033.027,E2 -28033.027} C_VEL
LIN {X 0,Y 106.183,Z 466.758,A -85,B 0,C 180,E1 -28035.355,E2 -28035.355} C_VEL
LIN {X 0,Y 109.882,Z 454.688,A -85,B 0,C 180,E1 -28037.349,E2 -28037.349} C_VEL
LIN {X 0,Y 112.501,Z 443.031,A -85,B 0,C 180,E1 -28038.727,E2 -28038.727} C_VEL
LIN {X 0,Y 114.688,Z 429.417,A -85,B 0,C 180,E1 -28039.584,E2 -28039.584} C_VEL
LIN {X 0,Y 117.351,Z 401.174,A -85,B 0,C 180,E1 -28040.77,E2 -28040.77} C_VEL
LIN {X 0,Y 113.941,Z 393.479,A -85,B 0,C 180,E1 -28044.379,E2 -28044.379} C_VEL
LIN {X 0,Y 110.408,Z 386.573,A -85,B 0,C 180,E1 -28048.703,E2 -28048.703} C_VEL
LIN {X 0,Y 107.985,Z 382.417,A -85,B 0,C 180,E1 -28052.195,E2 -28052.195} C_VEL
LIN {X 0,Y 106.483,Z 379.8,A -85,B 0,C 180,E1 -28054.744,E2 -28054.744} C_VEL
LIN {X 0,Y 104.435,Z 376.311,A -85,B 0,C 180,E1 -28058.979,E2 -28058.979} C_VEL
LIN {X 0,Y 102.265,Z 372.822,A -85,B 0,C 180,E1 -28065.575,E2 -28065.575} C_VEL
LIN {X 0,Y 101.982,Z 371.785,A -85,B 0,C 180,E1 -28067.163,E2 -28067.163} C_VEL
LIN {X 0,Y 101.199,Z 371.188,A -85,B 0,C 180,E1 -28076.018,E2 -28076.018} C_VEL
LIN {X 0,Y 101.706,Z 371.321,A -85,B 0,C 180,E1 -28080.743,E2 -28080.743} C_VEL
LIN {X 0,Y 102.303,Z 371.987,A -85,B 0,C 180,E1 -28083.693,E2 -28083.693} C_VEL
LIN {X 0,Y 104.012,Z 375.624,A -85,B 0,C 180,E1 -28089.48,E2 -28089.48} C_VEL
LIN {X 0,Y 104.849,Z 376.799,A -85,B 0,C 180,E1 -28091.42,E2 -28091.42} C_VEL
LIN {X 0,Y 107.373,Z 381.184,A -85,B 0,C 180,E1 -28096.274,E2 -28096.274} C_VEL
LIN {X 0,Y 109.748,Z 385.333,A -85,B 0,C 180,E1 -28099.89,E2 -28099.89} C_VEL
LIN {X 0,Y 112.611,Z 390.689,A -85,B 0,C 180,E1 -28103.567,E2 -28103.567} C_VEL
LIN {X 0,Y 114.715,Z 395.342,A -85,B 0,C 180,E1 -28106.004,E2 -28106.004} C_VEL
LIN {X 0,Y 116.926,Z 403.053,A -85,B 0,C 180,E1 -28108.619,E2 -28108.619} C_VEL
LIN {X 0,Y 117.184,Z 404.052,A -85,B 0,C 180,E1 -28108.917,E2 -28108.917} C_VEL
LIN {X 0,Y 113.884,Z 438.355,A -85,B 0,C 180,E1 -28110.443,E2 -28110.443} C_VEL
LIN {X 0,Y 111.321,Z 452.112,A -85,B 0,C 180,E1 -28111.51,E2 -28111.51} C_VEL
LIN {X 0,Y 107.885,Z 464.586,A -85,B 0,C 180,E1 -28112.999,E2 -28112.999} C_VEL
LIN {X 0,Y 103.181,Z 477.241,A -85,B 0,C 180,E1 -28115.184,E2 -28115.184} C_VEL
LIN {X 0,Y 98.036,Z 488.517,A -85,B 0,C 180,E1 -28117.953,E2 -28117.953} C_VEL
LIN {X 0,Y 92.69,Z 498.664,A -85,B 0,C 180,E1 -28121.523,E2 -28121.523} C_VEL
LIN {X 0,Y 86.694,Z 508.654,A -85,B 0,C 180,E1 -28126.448,E2 -28126.448} C_VEL
LIN {X 0,Y 82.787,Z 514.335,A -85,B 0,C 180,E1 -28130.068,E2 -28130.068} C_VEL
LIN {X 0,Y 80.124,Z 518.673,A -85,B 0,C 180,E1 -28133.7,E2 -28133.7} C_VEL
LIN {X 0,Y 75.598,Z 525.424,A -85,B 0,C 180,E1 -28140.79,E2 -28140.79} C_VEL
LIN {X 0,Y 71.842,Z 531.585,A -85,B 0,C 180,E1 -28149.981,E2 -28149.981} C_VEL
LIN {X 0,Y 70.209,Z 535.578,A -85,B 0,C 180,E1 -28158.455,E2 -28158.455} C_VEL
LIN {X 0,Y 69.779,Z 537.618,A -85,B 0,C 180,E1 -28164.223,E2 -28164.223} C_VEL
LIN {X 0,Y 69.883,Z 539.231,A -85,B 0,C 180,E1 -28170.003,E2 -28170.003} C_VEL
LIN {X 0,Y 69.774,Z 540.397,A -85,B 0,C 180,E1 -28175.784,E2 -28175.784} C_VEL
LIN {X 0,Y 70.209,Z 541.13,A -85,B 0,C 180,E1 -28181.552,E2 -28181.552} C_VEL
LIN {X 0,Y 72.936,Z 541.417,A -85,B 0,C 180,E1 -28192.673,E2 -28192.673} C_VEL
LIN {X 0,Y 75.187,Z 540.994,A -85,B 0,C 180,E1 -28197.867,E2 -28197.867} C_VEL
LIN {X 0,Y 78.136,Z 540.185,A -85,B 0,C 180,E1 -28202.664,E2 -28202.664} C_VEL
LIN {X 0,Y 85.483,Z 537.318,A -85,B 0,C 180,E1 -28211.129,E2 -28211.129} C_VEL
LIN {X 0,Y 92.062,Z 534.027,A -85,B 0,C 180,E1 -28216.601,E2 -28216.601} C_VEL
LIN {X 0,Y 99.193,Z 529.785,A -85,B 0,C 180,E1 -28221.205,E2 -28221.205} C_VEL
LIN {X 0,Y 108.443,Z 523.332,A -85,B 0,C 180,E1 -28225.723,E2 -28225.723} C_VEL
LIN {X 0,Y 116.873,Z 516.298,A -85,B 0,C 180,E1 -28228.973,E2 -28228.973} C_VEL
LIN {X 0,Y 125.661,Z 507.531,A -85,B 0,C 180,E1 -28231.75,E2 -28231.75} C_VEL
LIN {X 0,Y 133.931,Z 497.601,A -85,B 0,C 180,E1 -28233.981,E2 -28233.981} C_VEL
LIN {X 0,Y 140.867,Z 487.502,A -85,B 0,C 180,E1 -28235.578,E2 -28235.578} C_VEL
LIN {X 0,Y 147.206,Z 476.295,A -85,B 0,C 180,E1 -28236.789,E2 -28236.789} C_VEL
LIN {X 0,Y 152.515,Z 464.377,A -85,B 0,C 180,E1 -28237.745,E2 -28237.745} C_VEL
LIN {X 0,Y 156.673,Z 451.77,A -85,B 0,C 180,E1 -28238.498,E2 -28238.498} C_VEL
LIN {X 0,Y 159.429,Z 439.509,A -85,B 0,C 180,E1 -28239.024,E2 -28239.024} C_VEL
LIN {X 0,Y 158.307,Z 433.954,A -85,B 0,C 180,E1 -28241.894,E2 -28241.894} C_VEL
LIN {X 0,Y 157.311,Z 430.405,A -85,B 0,C 180,E1 -28244.451,E2 -28244.451} C_VEL
LIN {X 0,Y 155.758,Z 426.338,A -85,B 0,C 180,E1 -28249.602,E2 -28249.602} C_VEL
LIN {X 0,Y 155.109,Z 425.269,A -85,B 0,C 180,E1 -28254.8,E2 -28254.8} C_VEL
LIN {X 0,Y 155.152,Z 425.177,A -85,B 0,C 180,E1 -28256.507,E2 -28256.507} C_VEL
LIN {X 0,Y 155.253,Z 425.515,A -85,B 0,C 180,E1 -28257.952,E2 -28257.952} C_VEL
LIN {X 0,Y 155.42,Z 427.24,A -85,B 0,C 180,E1 -28260.041,E2 -28260.041} C_VEL
LIN {X 0,Y 155.592,Z 429.931,A -85,B 0,C 180,E1 -28262.004,E2 -28262.004} C_VEL
LIN {X 0,Y 156.305,Z 438.721,A -85,B 0,C 180,E1 -28267.11,E2 -28267.11} C_VEL
LIN {X 0,Y 156.921,Z 441.221,A -85,B 0,C 180,E1 -28269.099,E2 -28269.099} C_VEL
LIN {X 0,Y 153.81,Z 452.985,A -85,B 0,C 180,E1 -28269.717,E2 -28269.717} C_VEL
LIN {X 0,Y 149.534,Z 464.617,A -85,B 0,C 180,E1 -28270.497,E2 -28270.497} C_VEL
LIN {X 0,Y 144.339,Z 475.627,A -85,B 0,C 180,E1 -28271.587,E2 -28271.587} C_VEL
LIN {X 0,Y 137.919,Z 486.358,A -85,B 0,C 180,E1 -28272.948,E2 -28272.948} C_VEL
LIN {X 0,Y 130.786,Z 496.187,A -85,B 0,C 180,E1 -28274.699,E2 -28274.699} C_VEL
LIN {X 0,Y 122.241,Z 505.848,A -85,B 0,C 180,E1 -28276.995,E2 -28276.995} C_VEL
LIN {X 0,Y 113.798,Z 513.688,A -85,B 0,C 180,E1 -28279.637,E2 -28279.637} C_VEL
LIN {X 0,Y 104.976,Z 520.543,A -85,B 0,C 180,E1 -28282.994,E2 -28282.994} C_VEL
LIN {X 0,Y 95.237,Z 526.793,A -85,B 0,C 180,E1 -28287.679,E2 -28287.679} C_VEL
LIN {X 0,Y 87.464,Z 530.82,A -85,B 0,C 180,E1 -28292.463,E2 -28292.463} C_VEL
LIN {X 0,Y 80.43,Z 533.763,A -85,B 0,C 180,E1 -28298.144,E2 -28298.144} C_VEL
LIN {X 0,Y 76.194,Z 535.149,A -85,B 0,C 180,E1 -28302.443,E2 -28302.443} C_VEL
LIN {X 0,Y 69.195,Z 536.688,A -85,B 0,C 180,E1 -28312.45,E2 -28312.45} C_VEL
LIN {X 0,Y 66.593,Z 536.847,A -85,B 0,C 180,E1 -28318.148,E2 -28318.148} C_VEL
LIN {X 0,Y 64.548,Z 536.57,A -85,B 0,C 180,E1 -28324.178,E2 -28324.178} C_VEL
LIN {X 0,Y 62.472,Z 534.844,A -85,B 0,C 180,E1 -28336.994,E2 -28336.994} C_VEL
LIN {X 0,Y 62.484,Z 533.355,A -85,B 0,C 180,E1 -28343.539,E2 -28343.539} C_VEL
LIN {X 0,Y 63.521,Z 530.739,A -85,B 0,C 180,E1 -28351.988,E2 -28351.988} C_VEL
LIN {X 0,Y 66.014,Z 526.259,A -85,B 0,C 180,E1 -28362.29,E2 -28362.29} C_VEL
LIN {X 0,Y 70.503,Z 520.023,A -85,B 0,C 180,E1 -28371.947,E2 -28371.947} C_VEL
LIN {X 0,Y 75.535,Z 513.253,A -85,B 0,C 180,E1 -28379.237,E2 -28379.237} C_VEL
LIN {X 0,Y 81.594,Z 504.823,A -85,B 0,C 180,E1 -28385.545,E2 -28385.545} C_VEL
LIN {X 0,Y 87.255,Z 496.143,A -85,B 0,C 180,E1 -28390.114,E2 -28390.114} C_VEL
LIN {X 0,Y 93.43,Z 485.444,A -85,B 0,C 180,E1 -28394.087,E2 -28394.087} C_VEL
LIN {X 0,Y 98.688,Z 474.77,A -85,B 0,C 180,E1 -28396.878,E2 -28396.878} C_VEL
LIN {X 0,Y 103.318,Z 462.856,A -85,B 0,C 180,E1 -28399.175,E2 -28399.175} C_VEL
LIN {X 0,Y 106.821,Z 450.567,A -85,B 0,C 180,E1 -28400.998,E2 -28400.998} C_VEL
LIN {X 0,Y 109.525,Z 438.04,A -85,B 0,C 180,E1 -28402.138,E2 -28402.138} C_VEL
LIN {X 0,Y 111.433,Z 423.426,A -85,B 0,C 180,E1 -28402.843,E2 -28402.843} C_VEL
LIN {X 0,Y 113.299,Z 403.963,A -85,B 0,C 180,E1 -28403.64,E2 -28403.64} C_VEL
LIN {X 0,Y 110.093,Z 396.602,A -85,B 0,C 180,E1 -28407.587,E2 -28407.587} C_VEL
LIN {X 0,Y 106.79,Z 389.885,A -85,B 0,C 180,E1 -28412.451,E2 -28412.451} C_VEL
LIN {X 0,Y 104.692,Z 386.131,A -85,B 0,C 180,E1 -28416.248,E2 -28416.248} C_VEL
LIN {X 0,Y 102.929,Z 382.912,A -85,B 0,C 180,E1 -28420.344,E2 -28420.344} C_VEL
LIN {X 0,Y 101.071,Z 379.316,A -85,B 0,C 180,E1 -28427.045,E2 -28427.045} C_VEL
LIN {X 0,Y 100.944,Z 378.739,A -85,B 0,C 180,E1 -28427.944,E2 -28427.944} C_VEL
LIN {X 0,Y 100.327,Z 378.236,A -85,B 0,C 180,E1 -28435.984,E2 -28435.984} C_VEL
LIN {X 0,Y 100.958,Z 378.518,A -85,B 0,C 180,E1 -28441.496,E2 -28441.496} C_VEL
LIN {X 0,Y 101.233,Z 379.045,A -85,B 0,C 180,E1 -28442.985,E2 -28442.985} C_VEL
LIN {X 0,Y 103.38,Z 383.494,A -85,B 0,C 180,E1 -28450.253,E2 -28450.253} C_VEL
LIN {X 0,Y 105.645,Z 387.723,A -85,B 0,C 180,E1 -28455.053,E2 -28455.053} C_VEL
LIN {X 0,Y 108.403,Z 392.915,A -85,B 0,C 180,E1 -28459.53,E2 -28459.53} C_VEL
LIN {X 0,Y 111.4,Z 399.501,A -85,B 0,C 180,E1 -28463.592,E2 -28463.592} C_VEL
LIN {X 0,Y 113.168,Z 406.153,A -85,B 0,C 180,E1 -28466.014,E2 -28466.014} C_VEL
LIN {X 0,Y 110.011,Z 437.762,A -85,B 0,C 180,E1 -28467.404,E2 -28467.404} C_VEL
LIN {X 0,Y 107.336,Z 451.62,A -85,B 0,C 180,E1 -28468.43,E2 -28468.43} C_VEL
LIN {X 0,Y 103.816,Z 463.991,A -85,B 0,C 180,E1 -28469.851,E2 -28469.851} C_VEL
LIN {X 0,Y 99.262,Z 475.931,A -85,B 0,C 180,E1 -28471.834,E2 -28471.834} C_VEL
LIN {X 0,Y 93.839,Z 487.399,A -85,B 0,C 180,E1 -28474.534,E2 -28474.534} C_VEL
LIN {X 0,Y 88.089,Z 497.738,A -85,B 0,C 180,E1 -28478.019,E2 -28478.019} C_VEL
LIN {X 0,Y 81.666,Z 507.846,A -85,B 0,C 180,E1 -28482.993,E2 -28482.993} C_VEL
LIN {X 0,Y 76.124,Z 515.563,A -85,B 0,C 180,E1 -28488.275,E2 -28488.275} C_VEL
LIN {X 0,Y 71.011,Z 522.729,A -85,B 0,C 180,E1 -28495.318,E2 -28495.318} C_VEL
LIN {X 0,Y 67.351,Z 527.7,A -85,B 0,C 180,E1 -28501.998,E2 -28501.998} C_VEL
LIN {X 0,Y 64.37,Z 532.527,A -85,B 0,C 180,E1 -28510.884,E2 -28510.884} C_VEL
LIN {X 0,Y 62.881,Z 536.21,A -85,B 0,C 180,E1 -28520.352,E2 -28520.352} C_VEL
LIN {X 0,Y 62.788,Z 538.847,A -85,B 0,C 180,E1 -28530.003,E2 -28530.003} C_VEL
LIN {X 0,Y 62.723,Z 540.04,A -85,B 0,C 180,E1 -28536.437,E2 -28536.437} C_VEL
LIN {X 0,Y 63.259,Z 540.824,A -85,B 0,C 180,E1 -28542.841,E2 -28542.841} C_VEL
LIN {X 0,Y 66.417,Z 541.164,A -85,B 0,C 180,E1 -28555.044,E2 -28555.044} C_VEL
LIN {X 0,Y 68.966,Z 540.768,A -85,B 0,C 180,E1 -28560.635,E2 -28560.635} C_VEL
LIN {X 0,Y 72.241,Z 539.999,A -85,B 0,C 180,E1 -28565.715,E2 -28565.715} C_VEL
LIN {X 0,Y 75.99,Z 538.802,A -85,B 0,C 180,E1 -28570.349,E2 -28570.349} C_VEL
LIN {X 0,Y 82.512,Z 536.269,A -85,B 0,C 180,E1 -28576.388,E2 -28576.388} C_VEL
LIN {X 0,Y 89.741,Z 532.747,A -85,B 0,C 180,E1 -28581.552,E2 -28581.552} C_VEL
LIN {X 0,Y 97.598,Z 528.155,A -85,B 0,C 180,E1 -28585.908,E2 -28585.908} C_VEL
LIN {X 0,Y 107.487,Z 521.239,A -85,B 0,C 180,E1 -28590.04,E2 -28590.04} C_VEL
LIN {X 0,Y 116.379,Z 513.78,A -85,B 0,C 180,E1 -28592.968,E2 -28592.968} C_VEL
LIN {X 0,Y 123.976,Z 506.193,A -85,B 0,C 180,E1 -28595.098,E2 -28595.098} C_VEL
LIN {X 0,Y 131.79,Z 497.016,A -85,B 0,C 180,E1 -28596.913,E2 -28596.913} C_VEL
LIN {X 0,Y 138.903,Z 486.833,A -85,B 0,C 180,E1 -28598.392,E2 -28598.392} C_VEL
LIN {X 0,Y 145.382,Z 475.538,A -85,B 0,C 180,E1 -28599.493,E2 -28599.493} C_VEL
LIN {X 0,Y 150.576,Z 464.031,A -85,B 0,C 180,E1 -28600.337,E2 -28600.337} C_VEL
LIN {X 0,Y 154.732,Z 451.694,A -85,B 0,C 180,E1 -28601.024,E2 -28601.024} C_VEL
LIN {X 0,Y 156.866,Z 443.019,A -85,B 0,C 180,E1 -28601.384,E2 -28601.384} C_VEL
LIN {X 0,Y 156.15,Z 438.572,A -85,B 0,C 180,E1 -28604.081,E2 -28604.081} C_VEL
LIN {X 0,Y 155.693,Z 436.469,A -85,B 0,C 180,E1 -28605.791,E2 -28605.791} C_VEL
LIN {X 0,Y 154.666,Z 433.236,A -85,B 0,C 180,E1 -28610.189,E2 -28610.189} C_VEL
LIN {X 0,Y 154.167,Z 432.315,A -85,B 0,C 180,E1 -28614.769,E2 -28614.769} C_VEL
LIN {X 0,Y 154.349,Z 432.26,A -85,B 0,C 180,E1 -28618.043,E2 -28618.043} C_VEL
LIN {X 0,Y 154.804,Z 433.46,A -85,B 0,C 180,E1 -28621.12,E2 -28621.12} C_VEL
LIN {X 0,Y 155.74,Z 436.902,A -85,B 0,C 180,E1 -28625.34,E2 -28625.34} C_VEL
LIN {X 0,Y 156.305,Z 438.721,A -85,B 0,C 180,E1 -28627.11,E2 -28627.11} C_VEL
LIN {X 0,Y 156.241,Z 440.509,A -85,B 0,C 180,E1 -28627.72,E2 -28627.72} C_VEL
LIN {X 0,Y 155.684,Z 443.531,A -85,B 0,C 180,E1 -28628.052,E2 -28628.052} C_VEL
LIN {X 0,Y 154.324,Z 448.117,A -85,B 0,C 180,E1 -28627.983,E2 -28627.983} C_VEL
LIN {X 0,Y 151.156,Z 456.364,A -85,B 0,C 180,E1 -28627.388,E2 -28627.388} C_VEL
LIN {X 0,Y 150.102,Z 459.079,A -85,B 0,C 180,E1 -28627.431,E2 -28627.431} C_VEL
LIN {X 0,Y 145.228,Z 470.54,A -85,B 0,C 180,E1 -28628.347,E2 -28628.347} C_VEL
LIN {X 0,Y 138.944,Z 481.887,A -85,B 0,C 180,E1 -28629.476,E2 -28629.476} C_VEL
LIN {X 0,Y 131.564,Z 492.642,A -85,B 0,C 180,E1 -28631.013,E2 -28631.013} C_VEL
LIN {X 0,Y 124.284,Z 501.389,A -85,B 0,C 180,E1 -28632.719,E2 -28632.719} C_VEL
LIN {X 0,Y 116.296,Z 509.399,A -85,B 0,C 180,E1 -28634.777,E2 -28634.777} C_VEL
LIN {X 0,Y 106.913,Z 517.168,A -85,B 0,C 180,E1 -28637.601,E2 -28637.601} C_VEL
LIN {X 0,Y 97.741,Z 523.449,A -85,B 0,C 180,E1 -28641.07,E2 -28641.07} C_VEL
LIN {X 0,Y 89.25,Z 528.247,A -85,B 0,C 180,E1 -28645.096,E2 -28645.096} C_VEL
LIN {X 0,Y 81.139,Z 531.968,A -85,B 0,C 180,E1 -28649.98,E2 -28649.98} C_VEL
LIN {X 0,Y 76.134,Z 533.871,A -85,B 0,C 180,E1 -28653.815,E2 -28653.815} C_VEL
LIN {X 0,Y 71.482,Z 535.314,A -85,B 0,C 180,E1 -28658.132,E2 -28658.132} C_VEL
LIN {X 0,Y 63.581,Z 536.913,A -85,B 0,C 180,E1 -28668.451,E2 -28668.451} C_VEL
LIN {X 0,Y 60.547,Z 537.118,A -85,B 0,C 180,E1 -28674.519,E2 -28674.519} C_VEL
LIN {X 0,Y 58.097,Z 536.886,A -85,B 0,C 180,E1 -28681.057,E2 -28681.057} C_VEL
LIN {X 0,Y 55.452,Z 535.219,A -85,B 0,C 180,E1 -28695.313,E2 -28695.313} C_VEL
LIN {X 0,Y 55.341,Z 533.786,A -85,B 0,C 180,E1 -28702.7,E2 -28702.7} C_VEL
LIN {X 0,Y 56.546,Z 530.895,A -85,B 0,C 180,E1 -28713.256,E2 -28713.256} C_VEL
LIN {X 0,Y 59.103,Z 526.808,A -85,B 0,C 180,E1 -28723.754,E2 -28723.754} C_VEL
LIN {X 0,Y 63.987,Z 520.66,A -85,B 0,C 180,E1 -28734.319,E2 -28734.319} C_VEL
LIN {X 0,Y 69.449,Z 513.972,A -85,B 0,C 180,E1 -28742.088,E2 -28742.088} C_VEL
LIN {X 0,Y 75.954,Z 505.671,A -85,B 0,C 180,E1 -28748.647,E2 -28748.647} C_VEL
LIN {X 0,Y 81.964,Z 497.129,A -85,B 0,C 180,E1 -28753.307,E2 -28753.307} C_VEL
LIN {X 0,Y 88.493,Z 486.575,A -85,B 0,C 180,E1 -28757.271,E2 -28757.271} C_VEL
LIN {X 0,Y 93.973,Z 476.105,A -85,B 0,C 180,E1 -28760.043,E2 -28760.043} C_VEL
LIN {X 0,Y 98.859,Z 464.58,A -85,B 0,C 180,E1 -28762.264,E2 -28762.264} C_VEL
LIN {X 0,Y 102.896,Z 451.45,A -85,B 0,C 180,E1 -28764.197,E2 -28764.197} C_VEL
LIN {X 0,Y 105.747,Z 438.95,A -85,B 0,C 180,E1 -28765.328,E2 -28765.328} C_VEL
LIN {X 0,Y 107.603,Z 426.199,A -85,B 0,C 180,E1 -28765.946,E2 -28765.946} C_VEL
LIN {X 0,Y 109.527,Z 407.009,A -85,B 0,C 180,E1 -28766.7,E2 -28766.7} C_VEL
LIN {X 0,Y 106.839,Z 400.542,A -85,B 0,C 180,E1 -28770.589,E2 -28770.589} C_VEL
LIN {X 0,Y 104.335,Z 395.147,A -85,B 0,C 180,E1 -28774.942,E2 -28774.942} C_VEL
LIN {X 0,Y 102.812,Z 392.147,A -85,B 0,C 180,E1 -28778.183,E2 -28778.183} C_VEL
LIN {X 0,Y 101.542,Z 389.546,A -85,B 0,C 180,E1 -28781.592,E2 -28781.592} C_VEL
LIN {X 0,Y 99.906,Z 385.689,A -85,B 0,C 180,E1 -28788.846,E2 -28788.846} C_VEL
LIN {X 0,Y 99.455,Z 385.284,A -85,B 0,C 180,E1 -28795.948,E2 -28795.948} C_VEL
LIN {X 0,Y 100.082,Z 385.574,A -85,B 0,C 180,E1 -28801.509,E2 -28801.509} C_VEL
LIN {X 0,Y 101.998,Z 390.26,A -85,B 0,C 180,E1 -28809.169,E2 -28809.169} C_VEL
LIN {X 0,Y 103.914,Z 394.191,A -85,B 0,C 180,E1 -28813.693,E2 -28813.693} C_VEL
LIN {X 0,Y 106.173,Z 398.835,A -85,B 0,C 180,E1 -28817.797,E2 -28817.797} C_VEL
LIN {X 0,Y 108.567,Z 404.62,A -85,B 0,C 180,E1 -28821.479,E2 -28821.479} C_VEL
LIN {X 0,Y 109.456,Z 408.312,A -85,B 0,C 180,E1 -28822.909,E2 -28822.909} C_VEL
LIN {X 0,Y 106.302,Z 438.166,A -85,B 0,C 180,E1 -28824.204,E2 -28824.204} C_VEL
LIN {X 0,Y 103.573,Z 451.594,A -85,B 0,C 180,E1 -28825.166,E2 -28825.166} C_VEL
LIN {X 0,Y 99.724,Z 464.421,A -85,B 0,C 180,E1 -28826.607,E2 -28826.607} C_VEL
LIN {X 0,Y 94.971,Z 476.21,A -85,B 0,C 180,E1 -28828.512,E2 -28828.512} C_VEL
LIN {X 0,Y 89.287,Z 487.578,A -85,B 0,C 180,E1 -28831.136,E2 -28831.136} C_VEL
LIN {X 0,Y 83.219,Z 497.815,A -85,B 0,C 180,E1 -28834.578,E2 -28834.578} C_VEL
LIN {X 0,Y 76.975,Z 507.04,A -85,B 0,C 180,E1 -28839.103,E2 -28839.103} C_VEL
LIN {X 0,Y 71.119,Z 514.46,A -85,B 0,C 180,E1 -28844.024,E2 -28844.024} C_VEL
LIN {X 0,Y 67.077,Z 519.808,A -85,B 0,C 180,E1 -28849.097,E2 -28849.097} C_VEL
LIN {X 0,Y 62.703,Z 525.243,A -85,B 0,C 180,E1 -28855.92,E2 -28855.92} C_VEL
LIN {X 0,Y 58.618,Z 530.545,A -85,B 0,C 180,E1 -28865.193,E2 -28865.193} C_VEL
LIN {X 0,Y 56.302,Z 534.662,A -85,B 0,C 180,E1 -28875.547,E2 -28875.547} C_VEL
LIN {X 0,Y 55.635,Z 536.792,A -85,B 0,C 180,E1 -28882.747,E2 -28882.747} C_VEL
LIN {X 0,Y 55.685,Z 538.462,A -85,B 0,C 180,E1 -28890.004,E2 -28890.004} C_VEL
LIN {X 0,Y 55.657,Z 539.681,A -85,B 0,C 180,E1 -28897.258,E2 -28897.258} C_VEL
LIN {X 0,Y 56.334,Z 540.505,A -85,B 0,C 180,E1 -28904.452,E2 -28904.452} C_VEL
LIN {X 0,Y 57.826,Z 540.906,A -85,B 0,C 180,E1 -28911.387,E2 -28911.387} C_VEL
LIN {X 0,Y 62.943,Z 540.542,A -85,B 0,C 180,E1 -28923.941,E2 -28923.941} C_VEL
LIN {X 0,Y 66.59,Z 539.802,A -85,B 0,C 180,E1 -28929.294,E2 -28929.294} C_VEL
LIN {X 0,Y 70.711,Z 538.657,A -85,B 0,C 180,E1 -28934.089,E2 -28934.089} C_VEL
LIN {X 0,Y 75.343,Z 537.084,A -85,B 0,C 180,E1 -28938.269,E2 -28938.269} C_VEL
LIN {X 0,Y 81.406,Z 534.611,A -85,B 0,C 180,E1 -28942.819,E2 -28942.819} C_VEL
LIN {X 0,Y 90.968,Z 529.797,A -85,B 0,C 180,E1 -28948.197,E2 -28948.197} C_VEL
LIN {X 0,Y 101.116,Z 523.483,A -85,B 0,C 180,E1 -28952.4,E2 -28952.4} C_VEL
LIN {X 0,Y 110.237,Z 516.634,A -85,B 0,C 180,E1 -28955.3,E2 -28955.3} C_VEL
LIN {X 0,Y 118.025,Z 509.663,A -85,B 0,C 180,E1 -28957.367,E2 -28957.367} C_VEL
LIN {X 0,Y 125.963,Z 501.29,A -85,B 0,C 180,E1 -28959.159,E2 -28959.159} C_VEL
LIN {X 0,Y 134.029,Z 490.986,A -85,B 0,C 180,E1 -28960.712,E2 -28960.712} C_VEL
LIN {X 0,Y 140.584,Z 480.802,A -85,B 0,C 180,E1 -28961.778,E2 -28961.778} C_VEL
LIN {X 0,Y 146.365,Z 469.687,A -85,B 0,C 180,E1 -28962.621,E2 -28962.621} C_VEL
LIN {X 0,Y 150.995,Z 458.23,A -85,B 0,C 180,E1 -28963.284,E2 -28963.284} C_VEL
LIN {X 0,Y 154.418,Z 446.725,A -85,B 0,C 180,E1 -28963.812,E2 -28963.812} C_VEL
LIN {X 0,Y 153.988,Z 443.093,A -85,B 0,C 180,E1 -28966.473,E2 -28966.473} C_VEL
LIN {X 0,Y 153.283,Z 440.081,A -85,B 0,C 180,E1 -28970.765,E2 -28970.765} C_VEL
LIN {X 0,Y 152.918,Z 439.313,A -85,B 0,C 180,E1 -28974.726,E2 -28974.726} C_VEL
LIN {X 0,Y 153.106,Z 439.362,A -85,B 0,C 180,E1 -28978.356,E2 -28978.356} C_VEL
LIN {X 0,Y 153.321,Z 440.296,A -85,B 0,C 180,E1 -28980.59,E2 -28980.59} C_VEL
LIN {X 0,Y 153.973,Z 443.743,A -85,B 0,C 180,E1 -28984.909,E2 -28984.909} C_VEL
LIN {X 0,Y 154.331,Z 445.772,A -85,B 0,C 180,E1 -28986.774,E2 -28986.774} C_VEL
LIN {X 0,Y 150.102,Z 459.079,A -85,B 0,C 180,E1 -28987.431,E2 -28987.431} C_VEL
LIN {X 0,Y 147.816,Z 464.551,A -85,B 0,C 180,E1 -28987.532,E2 -28987.532} C_VEL
LIN {X 0,Y 143.159,Z 473.286,A -85,B 0,C 180,E1 -28987.102,E2 -28987.102} C_VEL
LIN {X 0,Y 137.849,Z 481.608,A -85,B 0,C 180,E1 -28986.781,E2 -28986.781} C_VEL
LIN {X 0,Y 134.531,Z 486.42,A -85,B 0,C 180,E1 -28987.098,E2 -28987.098} C_VEL
LIN {X 0,Y 127.871,Z 495.298,A -85,B 0,C 180,E1 -28988.379,E2 -28988.379} C_VEL
LIN {X 0,Y 119.45,Z 504.579,A -85,B 0,C 180,E1 -28990.166,E2 -28990.166} C_VEL
LIN {X 0,Y 109.769,Z 513.313,A -85,B 0,C 180,E1 -28992.471,E2 -28992.471} C_VEL
LIN {X 0,Y 100.191,Z 520.346,A -85,B 0,C 180,E1 -28995.306,E2 -28995.306} C_VEL
LIN {X 0,Y 89.403,Z 526.747,A -85,B 0,C 180,E1 -28999.377,E2 -28999.377} C_VEL
LIN {X 0,Y 80.578,Z 530.912,A -85,B 0,C 180,E1 -29003.675,E2 -29003.675} C_VEL
LIN {X 0,Y 72.105,Z 534.052,A -85,B 0,C 180,E1 -29009.165,E2 -29009.165} C_VEL
LIN {X 0,Y 67.233,Z 535.478,A -85,B 0,C 180,E1 -29013.249,E2 -29013.249} C_VEL
LIN {X 0,Y 58.339,Z 537.14,A -85,B 0,C 180,E1 -29023.709,E2 -29023.709} C_VEL
LIN {X 0,Y 54.48,Z 537.386,A -85,B 0,C 180,E1 -29030.714,E2 -29030.714} C_VEL
LIN {X 0,Y 49.735,Z 536.592,A -85,B 0,C 180,E1 -29044.913,E2 -29044.913} C_VEL
LIN {X 0,Y 48.505,Z 535.592,A -85,B 0,C 180,E1 -29053.15,E2 -29053.15} C_VEL
LIN {X 0,Y 48.207,Z 534.196,A -85,B 0,C 180,E1 -29061.613,E2 -29061.613} C_VEL
LIN {X 0,Y 49.224,Z 531.821,A -85,B 0,C 180,E1 -29071.958,E2 -29071.958} C_VEL
LIN {X 0,Y 52.244,Z 527.334,A -85,B 0,C 180,E1 -29085.603,E2 -29085.603} C_VEL
LIN {X 0,Y 56.733,Z 522.27,A -85,B 0,C 180,E1 -29095.69,E2 -29095.69} C_VEL
LIN {X 0,Y 62.523,Z 515.909,A -85,B 0,C 180,E1 -29104.192,E2 -29104.192} C_VEL
LIN {X 0,Y 69.308,Z 507.965,A -85,B 0,C 180,E1 -29111.228,E2 -29111.228} C_VEL
LIN {X 0,Y 76.96,Z 498.08,A -85,B 0,C 180,E1 -29116.928,E2 -29116.928} C_VEL
LIN {X 0,Y 83.863,Z 487.684,A -85,B 0,C 180,E1 -29120.816,E2 -29120.816} C_VEL
LIN {X 0,Y 89.577,Z 477.401,A -85,B 0,C 180,E1 -29123.527,E2 -29123.527} C_VEL
LIN {X 0,Y 94.707,Z 466.152,A -85,B 0,C 180,E1 -29125.64,E2 -29125.64} C_VEL
LIN {X 0,Y 98.988,Z 453.543,A -85,B 0,C 180,E1 -29127.464,E2 -29127.464} C_VEL
LIN {X 0,Y 101.825,Z 442.083,A -85,B 0,C 180,E1 -29128.599,E2 -29128.599} C_VEL
LIN {X 0,Y 104.149,Z 428.288,A -85,B 0,C 180,E1 -29129.282,E2 -29129.282} C_VEL
LIN {X 0,Y 106.037,Z 410.851,A -85,B 0,C 180,E1 -29129.879,E2 -29129.879} C_VEL
LIN {X 0,Y 105.89,Z 409.707,A -85,B 0,C 180,E1 -29130.237,E2 -29130.237} C_VEL
LIN {X 0,Y 103.473,Z 403.572,A -85,B 0,C 180,E1 -29134.567,E2 -29134.567} C_VEL
LIN {X 0,Y 101.422,Z 398.905,A -85,B 0,C 180,E1 -29139.204,E2 -29139.204} C_VEL
LIN {X 0,Y 100.156,Z 396.112,A -85,B 0,C 180,E1 -29143.034,E2 -29143.034} C_VEL
LIN {X 0,Y 98.895,Z 392.622,A -85,B 0,C 180,E1 -29149.767,E2 -29149.767} C_VEL
LIN {X 0,Y 98.962,Z 392.398,A -85,B 0,C 180,E1 -29160.001,E2 -29160.001} C_VEL
LIN {X 0,Y 99.263,Z 393.596,A -85,B 0,C 180,E1 -29162.346,E2 -29162.346} C_VEL
LIN {X 0,Y 100.652,Z 396.95,A -85,B 0,C 180,E1 -29168.028,E2 -29168.028} C_VEL
LIN {X 0,Y 102.397,Z 401.003,A -85,B 0,C 180,E1 -29172.638,E2 -29172.638} C_VEL
LIN {X 0,Y 104.573,Z 406.099,A -85,B 0,C 180,E1 -29176.974,E2 -29176.974} C_VEL
LIN {X 0,Y 105.933,Z 410.12,A -85,B 0,C 180,E1 -29179.374,E2 -29179.374} C_VEL
LIN {X 0,Y 106.083,Z 410.786,A -85,B 0,C 180,E1 -29179.656,E2 -29179.656} C_VEL
LIN {X 0,Y 103.033,Z 437.966,A -85,B 0,C 180,E1 -29180.75,E2 -29180.75} C_VEL
LIN {X 0,Y 100.164,Z 451.559,A -85,B 0,C 180,E1 -29181.67,E2 -29181.67} C_VEL
LIN {X 0,Y 96.349,Z 463.809,A -85,B 0,C 180,E1 -29182.948,E2 -29182.948} C_VEL
LIN {X 0,Y 91.026,Z 476.471,A -85,B 0,C 180,E1 -29184.886,E2 -29184.886} C_VEL
LIN {X 0,Y 85.083,Z 487.745,A -85,B 0,C 180,E1 -29187.388,E2 -29187.388} C_VEL
LIN {X 0,Y 78.685,Z 497.879,A -85,B 0,C 180,E1 -29190.725,E2 -29190.725} C_VEL
LIN {X 0,Y 71.376,Z 507.874,A -85,B 0,C 180,E1 -29195.682,E2 -29195.682} C_VEL
LIN {X 0,Y 65.099,Z 515.269,A -85,B 0,C 180,E1 -29200.918,E2 -29200.918} C_VEL
LIN {X 0,Y 59.765,Z 521.449,A -85,B 0,C 180,E1 -29207.461,E2 -29207.461} C_VEL
LIN {X 0,Y 55.149,Z 526.567,A -85,B 0,C 180,E1 -29215.013,E2 -29215.013} C_VEL
LIN {X 0,Y 51.065,Z 531.52,A -85,B 0,C 180,E1 -29225.619,E2 -29225.619} C_VEL
LIN {X 0,Y 48.919,Z 535.328,A -85,B 0,C 180,E1 -29237.56,E2 -29237.56} C_VEL
LIN {X 0,Y 48.579,Z 538.078,A -85,B 0,C 180,E1 -29250.004,E2 -29250.004} C_VEL
LIN {X 0,Y 48.608,Z 539.323,A -85,B 0,C 180,E1 -29258.318,E2 -29258.318} C_VEL
LIN {X 0,Y 49.479,Z 540.174,A -85,B 0,C 180,E1 -29266.508,E2 -29266.508} C_VEL
LIN {X 0,Y 51.255,Z 540.626,A -85,B 0,C 180,E1 -29274.294,E2 -29274.294} C_VEL
LIN {X 0,Y 57.177,Z 540.318,A -85,B 0,C 180,E1 -29287.926,E2 -29287.926} C_VEL
LIN {X 0,Y 65.783,Z 538.507,A -85,B 0,C 180,E1 -29298.408,E2 -29298.408} C_VEL
LIN {X 0,Y 70.796,Z 536.972,A -85,B 0,C 180,E1 -29302.58,E2 -29302.58} C_VEL
LIN {X 0,Y 78.819,Z 533.905,A -85,B 0,C 180,E1 -29307.895,E2 -29307.895} C_VEL
LIN {X 0,Y 87.428,Z 529.81,A -85,B 0,C 180,E1 -29312.163,E2 -29312.163} C_VEL
LIN {X 0,Y 98.029,Z 523.565,A -85,B 0,C 180,E1 -29316.08,E2 -29316.08} C_VEL
LIN {X 0,Y 107.472,Z 516.792,A -85,B 0,C 180,E1 -29318.73,E2 -29318.73} C_VEL
LIN {X 0,Y 115.484,Z 509.908,A -85,B 0,C 180,E1 -29320.613,E2 -29320.613} C_VEL
LIN {X 0,Y 123.624,Z 501.638,A -85,B 0,C 180,E1 -29322.223,E2 -29322.223} C_VEL
LIN {X 0,Y 131.864,Z 491.527,A -85,B 0,C 180,E1 -29323.611,E2 -29323.611} C_VEL
LIN {X 0,Y 138.539,Z 481.515,A -85,B 0,C 180,E1 -29324.552,E2 -29324.552} C_VEL
LIN {X 0,Y 144.415,Z 470.633,A -85,B 0,C 180,E1 -29325.292,E2 -29325.292} C_VEL
LIN {X 0,Y 149.488,Z 458.53,A -85,B 0,C 180,E1 -29325.924,E2 -29325.924} C_VEL
LIN {X 0,Y 151.993,Z 450.744,A -85,B 0,C 180,E1 -29326.295,E2 -29326.295} C_VEL
LIN {X 0,Y 151.852,Z 449.344,A -85,B 0,C 180,E1 -29327.64,E2 -29327.64} C_VEL
LIN {X 0,Y 151.513,Z 446.832,A -85,B 0,C 180,E1 -29331.329,E2 -29331.329} C_VEL
LIN {X 0,Y 151.361,Z 446.071,A -85,B 0,C 180,E1 -29337.338,E2 -29337.338} C_VEL
LIN {X 0,Y 151.479,Z 446.994,A -85,B 0,C 180,E1 -29340,E2 -29340} C_VEL
LIN {X 0,Y 151.782,Z 450.043,A -85,B 0,C 180,E1 -29343.984,E2 -29343.984} C_VEL
LIN {X 0,Y 151.817,Z 450.347,A -85,B 0,C 180,E1 -29344.315,E2 -29344.315} C_VEL
LIN {X 0,Y 147.392,Z 462.679,A -85,B 0,C 180,E1 -29344.958,E2 -29344.958} C_VEL
LIN {X 0,Y 141.332,Z 475.416,A -85,B 0,C 180,E1 -29345.985,E2 -29345.985} C_VEL
LIN {X 0,Y 134.531,Z 486.42,A -85,B 0,C 180,E1 -29347.098,E2 -29347.098} C_VEL
LIN {X 0,Y 130.992,Z 491.176,A -85,B 0,C 180,E1 -29347.468,E2 -29347.468} C_VEL
LIN {X 0,Y 124.378,Z 498.617,A -85,B 0,C 180,E1 -29347.333,E2 -29347.333} C_VEL
LIN {X 0,Y 117.265,Z 505.463,A -85,B 0,C 180,E1 -29347.245,E2 -29347.245} C_VEL
LIN {X 0,Y 112.963,Z 509.297,A -85,B 0,C 180,E1 -29347.767,E2 -29347.767} C_VEL
LIN {X 0,Y 103.454,Z 516.882,A -85,B 0,C 180,E1 -29349.915,E2 -29349.915} C_VEL
LIN {X 0,Y 93.653,Z 523.245,A -85,B 0,C 180,E1 -29352.686,E2 -29352.686} C_VEL
LIN {X 0,Y 84.109,Z 528.267,A -85,B 0,C 180,E1 -29356.065,E2 -29356.065} C_VEL
LIN {X 0,Y 74.922,Z 532.12,A -85,B 0,C 180,E1 -29360.269,E2 -29360.269} C_VEL
LIN {X 0,Y 68.029,Z 534.417,A -85,B 0,C 180,E1 -29364.408,E2 -29364.408} C_VEL
LIN {X 0,Y 58.307,Z 536.709,A -85,B 0,C 180,E1 -29372.457,E2 -29372.457} C_VEL
LIN {X 0,Y 49.403,Z 537.633,A -85,B 0,C 180,E1 -29384.655,E2 -29384.655} C_VEL
LIN {X 0,Y 45.935,Z 537.504,A -85,B 0,C 180,E1 -29392.261,E2 -29392.261} C_VEL
LIN {X 0,Y 43.301,Z 536.934,A -85,B 0,C 180,E1 -29400.857,E2 -29400.857} C_VEL
LIN {X 0,Y 41.662,Z 535.962,A -85,B 0,C 180,E1 -29410.277,E2 -29410.277} C_VEL
LIN {X 0,Y 41.093,Z 534.596,A -85,B 0,C 180,E1 -29420.147,E2 -29420.147} C_VEL
LIN {X 0,Y 42.249,Z 531.987,A -85,B 0,C 180,E1 -29433.571,E2 -29433.571} C_VEL
LIN {X 0,Y 45.457,Z 527.852,A -85,B 0,C 180,E1 -29448.007,E2 -29448.007} C_VEL
LIN {X 0,Y 50.421,Z 522.859,A -85,B 0,C 180,E1 -29459.194,E2 -29459.194} C_VEL
LIN {X 0,Y 56.792,Z 516.594,A -85,B 0,C 180,E1 -29468.22,E2 -29468.22} C_VEL
LIN {X 0,Y 64.143,Z 508.76,A -85,B 0,C 180,E1 -29475.408,E2 -29475.408} C_VEL
LIN {X 0,Y 72.304,Z 498.983,A -85,B 0,C 180,E1 -29481.036,E2 -29481.036} C_VEL
LIN {X 0,Y 79.571,Z 488.787,A -85,B 0,C 180,E1 -29484.779,E2 -29484.779} C_VEL
LIN {X 0,Y 86.324,Z 477.255,A -85,B 0,C 180,E1 -29487.631,E2 -29487.631} C_VEL
LIN {X 0,Y 91.661,Z 465.916,A -85,B 0,C 180,E1 -29489.601,E2 -29489.601} C_VEL
LIN {X 0,Y 95.769,Z 454.359,A -85,B 0,C 180,E1 -29491.162,E2 -29491.162} C_VEL
LIN {X 0,Y 98.946,Z 442.091,A -85,B 0,C 180,E1 -29492.292,E2 -29492.292} C_VEL
LIN {X 0,Y 101.3,Z 428.452,A -85,B 0,C 180,E1 -29492.901,E2 -29492.901} C_VEL
LIN {X 0,Y 102.931,Z 413.461,A -85,B 0,C 180,E1 -29493.441,E2 -29493.441} C_VEL
LIN {X 0,Y 100.982,Z 408.039,A -85,B 0,C 180,E1 -29497.766,E2 -29497.766} C_VEL
LIN {X 0,Y 99.696,Z 404.794,A -85,B 0,C 180,E1 -29501.372,E2 -29501.372} C_VEL
LIN {X 0,Y 98.894,Z 402.793,A -85,B 0,C 180,E1 -29504.28,E2 -29504.28} C_VEL
LIN {X 0,Y 97.906,Z 399.592,A -85,B 0,C 180,E1 -29510.706,E2 -29510.706} C_VEL
LIN {X 0,Y 97.837,Z 399.408,A -85,B 0,C 180,E1 -29517.942,E2 -29517.942} C_VEL
LIN {X 0,Y 98.109,Z 399.887,A -85,B 0,C 180,E1 -29520.475,E2 -29520.475} C_VEL
LIN {X 0,Y 99.294,Z 403.535,A -85,B 0,C 180,E1 -29526.675,E2 -29526.675} C_VEL
LIN {X 0,Y 100.901,Z 407.71,A -85,B 0,C 180,E1 -29531.496,E2 -29531.496} C_VEL
LIN {X 0,Y 102.692,Z 412.63,A -85,B 0,C 180,E1 -29535.545,E2 -29535.545} C_VEL
LIN {X 0,Y 102.99,Z 413.548,A -85,B 0,C 180,E1 -29536.154,E2 -29536.154} C_VEL
LIN {X 0,Y 100.127,Z 437.952,A -85,B 0,C 180,E1 -29537.106,E2 -29537.106} C_VEL
LIN {X 0,Y 97.09,Z 451.728,A -85,B 0,C 180,E1 -29537.965,E2 -29537.965} C_VEL
LIN {X 0,Y 92.998,Z 464.169,A -85,B 0,C 180,E1 -29539.163,E2 -29539.163} C_VEL
LIN {X 0,Y 87.476,Z 476.705,A -85,B 0,C 180,E1 -29540.946,E2 -29540.946} C_VEL
LIN {X 0,Y 81.279,Z 487.878,A -85,B 0,C 180,E1 -29543.269,E2 -29543.269} C_VEL
LIN {X 0,Y 74.549,Z 497.924,A -85,B 0,C 180,E1 -29546.423,E2 -29546.423} C_VEL
LIN {X 0,Y 67.461,Z 507.045,A -85,B 0,C 180,E1 -29550.75,E2 -29550.75} C_VEL
LIN {X 0,Y 60.592,Z 514.522,A -85,B 0,C 180,E1 -29555.723,E2 -29555.723} C_VEL
LIN {X 0,Y 55.853,Z 519.663,A -85,B 0,C 180,E1 -29560.983,E2 -29560.983} C_VEL
LIN {X 0,Y 49.471,Z 525.989,A -85,B 0,C 180,E1 -29570.268,E2 -29570.268} C_VEL
LIN {X 0,Y 44.658,Z 531.009,A -85,B 0,C 180,E1 -29581.834,E2 -29581.834} C_VEL
LIN {X 0,Y 41.994,Z 534.881,A -85,B 0,C 180,E1 -29595.467,E2 -29595.467} C_VEL
LIN {X 0,Y 41.469,Z 537.689,A -85,B 0,C 180,E1 -29610.005,E2 -29610.005} C_VEL
LIN {X 0,Y 41.597,Z 538.962,A -85,B 0,C 180,E1 -29619.732,E2 -29619.732} C_VEL
LIN {X 0,Y 44.841,Z 540.333,A -85,B 0,C 180,E1 -29638.052,E2 -29638.052} C_VEL
LIN {X 0,Y 51.753,Z 540.094,A -85,B 0,C 180,E1 -29652.77,E2 -29652.77} C_VEL
LIN {X 0,Y 61.29,Z 538.343,A -85,B 0,C 180,E1 -29663.391,E2 -29663.391} C_VEL
LIN {X 0,Y 66.707,Z 536.861,A -85,B 0,C 180,E1 -29667.447,E2 -29667.447} C_VEL
LIN {X 0,Y 75.274,Z 533.849,A -85,B 0,C 180,E1 -29672.5,E2 -29672.5} C_VEL
LIN {X 0,Y 84.346,Z 529.814,A -85,B 0,C 180,E1 -29676.433,E2 -29676.433} C_VEL
LIN {X 0,Y 95.374,Z 523.647,A -85,B 0,C 180,E1 -29679.977,E2 -29679.977} C_VEL
LIN {X 0,Y 105.105,Z 516.951,A -85,B 0,C 180,E1 -29682.34,E2 -29682.34} C_VEL
LIN {X 0,Y 114.986,Z 508.67,A -85,B 0,C 180,E1 -29684.294,E2 -29684.294} C_VEL
LIN {X 0,Y 123.302,Z 500.19,A -85,B 0,C 180,E1 -29685.694,E2 -29685.694} C_VEL
LIN {X 0,Y 130.882,Z 490.9,A -85,B 0,C 180,E1 -29686.725,E2 -29686.725} C_VEL
LIN {X 0,Y 138.53,Z 479.384,A -85,B 0,C 180,E1 -29687.585,E2 -29687.585} C_VEL
LIN {X 0,Y 144.621,Z 467.786,A -85,B 0,C 180,E1 -29688.219,E2 -29688.219} C_VEL
LIN {X 0,Y 149.159,Z 456.505,A -85,B 0,C 180,E1 -29688.697,E2 -29688.697} C_VEL
LIN {X 0,Y 149.452,Z 455.415,A -85,B 0,C 180,E1 -29688.94,E2 -29688.94} C_VEL
LIN {X 0,Y 149.376,Z 453.49,A -85,B 0,C 180,E1 -29691.885,E2 -29691.885} C_VEL
LIN {X 0,Y 149.296,Z 452.861,A -85,B 0,C 180,E1 -29697.302,E2 -29697.302} C_VEL
LIN {X 0,Y 149.288,Z 453.979,A -85,B 0,C 180,E1 -29700,E2 -29700} C_VEL
LIN {X 0,Y 149.287,Z 455.163,A -85,B 0,C 180,E1 -29701.69,E2 -29701.69} C_VEL
LIN {X 0,Y 148.99,Z 456.171,A -85,B 0,C 180,E1 -29701.931,E2 -29701.931} C_VEL
LIN {X 0,Y 144.874,Z 466.321,A -85,B 0,C 180,E1 -29702.442,E2 -29702.442} C_VEL
LIN {X 0,Y 139.033,Z 477.597,A -85,B 0,C 180,E1 -29703.286,E2 -29703.286} C_VEL
LIN {X 0,Y 132.848,Z 487.195,A -85,B 0,C 180,E1 -29704.167,E2 -29704.167} C_VEL
LIN {X 0,Y 125.312,Z 496.838,A -85,B 0,C 180,E1 -29705.436,E2 -29705.436} C_VEL
LIN {X 0,Y 116.343,Z 506.243,A -85,B 0,C 180,E1 -29707.081,E2 -29707.081} C_VEL
LIN {X 0,Y 112.963,Z 509.297,A -85,B 0,C 180,E1 -29707.767,E2 -29707.767} C_VEL
LIN {X 0,Y 108.477,Z 512.975,A -85,B 0,C 180,E1 -29708.368,E2 -29708.368} C_VEL
LIN {X 0,Y 100.287,Z 518.582,A -85,B 0,C 180,E1 -29708.551,E2 -29708.551} C_VEL
LIN {X 0,Y 91.726,Z 523.575,A -85,B 0,C 180,E1 -29708.869,E2 -29708.869} C_VEL
LIN {X 0,Y 86.685,Z 526.179,A -85,B 0,C 180,E1 -29709.845,E2 -29709.845} C_VEL
LIN {X 0,Y 75.907,Z 530.999,A -85,B 0,C 180,E1 -29713.542,E2 -29713.542} C_VEL
LIN {X 0,Y 64.422,Z 534.796,A -85,B 0,C 180,E1 -29719.103,E2 -29719.103} C_VEL
LIN {X 0,Y 54.738,Z 536.906,A -85,B 0,C 180,E1 -29725.998,E2 -29725.998} C_VEL
LIN {X 0,Y 44.59,Z 537.889,A -85,B 0,C 180,E1 -29737.987,E2 -29737.987} C_VEL
LIN {X 0,Y 40.449,Z 537.792,A -85,B 0,C 180,E1 -29745.966,E2 -29745.966} C_VEL
LIN {X 0,Y 37.138,Z 537.277,A -85,B 0,C 180,E1 -29755.402,E2 -29755.402} C_VEL
LIN {X 0,Y 34.936,Z 536.334,A -85,B 0,C 180,E1 -29766.269,E2 -29766.269} C_VEL
LIN {X 0,Y 34.01,Z 534.997,A -85,B 0,C 180,E1 -29778.068,E2 -29778.068} C_VEL
LIN {X 0,Y 35.33,Z 532.129,A -85,B 0,C 180,E1 -29795.953,E2 -29795.953} C_VEL
LIN {X 0,Y 38.776,Z 528.37,A -85,B 0,C 180,E1 -29811.247,E2 -29811.247} C_VEL
LIN {X 0,Y 44.339,Z 523.449,A -85,B 0,C 180,E1 -29823.689,E2 -29823.689} C_VEL
LIN {X 0,Y 51.405,Z 517.258,A -85,B 0,C 180,E1 -29833.118,E2 -29833.118} C_VEL
LIN {X 0,Y 59.381,Z 509.554,A -85,B 0,C 180,E1 -29840.284,E2 -29840.284} C_VEL
LIN {X 0,Y 68.072,Z 499.882,A -85,B 0,C 180,E1 -29845.679,E2 -29845.679} C_VEL
LIN {X 0,Y 75.724,Z 489.87,A -85,B 0,C 180,E1 -29849.141,E2 -29849.141} C_VEL
LIN {X 0,Y 82.746,Z 478.538,A -85,B 0,C 180,E1 -29851.781,E2 -29851.781} C_VEL
LIN {X 0,Y 88.305,Z 467.433,A -85,B 0,C 180,E1 -29853.548,E2 -29853.548} C_VEL
LIN {X 0,Y 92.982,Z 455.156,A -85,B 0,C 180,E1 -29855.088,E2 -29855.088} C_VEL
LIN {X 0,Y 96.25,Z 443.229,A -85,B 0,C 180,E1 -29856.13,E2 -29856.13} C_VEL
LIN {X 0,Y 98.68,Z 430.027,A -85,B 0,C 180,E1 -29856.676,E2 -29856.676} C_VEL
LIN {X 0,Y 100.156,Z 417.005,A -85,B 0,C 180,E1 -29857.151,E2 -29857.151} C_VEL
LIN {X 0,Y 98.926,Z 413.12,A -85,B 0,C 180,E1 -29860.683,E2 -29860.683} C_VEL
LIN {X 0,Y 97.712,Z 409.518,A -85,B 0,C 180,E1 -29865.42,E2 -29865.42} C_VEL
LIN {X 0,Y 96.989,Z 406.605,A -85,B 0,C 180,E1 -29871.143,E2 -29871.143} C_VEL
LIN {X 0,Y 97.061,Z 406.555,A -85,B 0,C 180,E1 -29878.963,E2 -29878.963} C_VEL
LIN {X 0,Y 97.994,Z 410.084,A -85,B 0,C 180,E1 -29885.273,E2 -29885.273} C_VEL
LIN {X 0,Y 99.392,Z 414.319,A -85,B 0,C 180,E1 -29890.182,E2 -29890.182} C_VEL
LIN {X 0,Y 100.249,Z 417.078,A -85,B 0,C 180,E1 -29892.53,E2 -29892.53} C_VEL
LIN {X 0,Y 97.575,Z 438.335,A -85,B 0,C 180,E1 -29893.272,E2 -29893.272} C_VEL
LIN {X 0,Y 94.611,Z 451.303,A -85,B 0,C 180,E1 -29894.002,E2 -29894.002} C_VEL
LIN {X 0,Y 90.502,Z 463.534,A -85,B 0,C 180,E1 -29895.03,E2 -29895.03} C_VEL
LIN {X 0,Y 85.164,Z 475.33,A -85,B 0,C 180,E1 -29896.409,E2 -29896.409} C_VEL
LIN {X 0,Y 78.75,Z 486.737,A -85,B 0,C 180,E1 -29898.529,E2 -29898.529} C_VEL
LIN {X 0,Y 72.418,Z 495.932,A -85,B 0,C 180,E1 -29900.931,E2 -29900.931} C_VEL
LIN {X 0,Y 65.575,Z 504.532,A -85,B 0,C 180,E1 -29904.368,E2 -29904.368} C_VEL
LIN {X 0,Y 58.114,Z 512.491,A -85,B 0,C 180,E1 -29908.931,E2 -29908.931} C_VEL
LIN {X 0,Y 54.055,Z 516.514,A -85,B 0,C 180,E1 -29912.38,E2 -29912.38} C_VEL
LIN {X 0,Y 46.515,Z 523.411,A -85,B 0,C 180,E1 -29920.943,E2 -29920.943} C_VEL
LIN {X 0,Y 40.171,Z 528.92,A -85,B 0,C 180,E1 -29932.249,E2 -29932.249} C_VEL
LIN {X 0,Y 35.977,Z 533.231,A -85,B 0,C 180,E1 -29947.009,E2 -29947.009} C_VEL
LIN {X 0,Y 34.567,Z 535.503,A -85,B 0,C 180,E1 -29958.275,E2 -29958.275} C_VEL
LIN {X 0,Y 34.378,Z 537.3,A -85,B 0,C 180,E1 -29970.006,E2 -29970.006} C_VEL
LIN {X 0,Y 34.611,Z 538.601,A -85,B 0,C 180,E1 -29981.722,E2 -29981.722} C_VEL
LIN {X 0,Y 38.688,Z 540.028,A -85,B 0,C 180,E1 -30003.029,E2 -30003.029} C_VEL
LIN {X 0,Y 42.303,Z 540.154,A -85,B 0,C 180,E1 -30011.653,E2 -30011.653} C_VEL
LIN {X 0,Y 51.858,Z 539.213,A -85,B 0,C 180,E1 -30024.41,E2 -30024.41} C_VEL
LIN {X 0,Y 63.153,Z 536.744,A -85,B 0,C 180,E1 -30032.915,E2 -30032.915} C_VEL
LIN {X 0,Y 72.264,Z 533.779,A -85,B 0,C 180,E1 -30037.511,E2 -30037.511} C_VEL
LIN {X 0,Y 81.76,Z 529.801,A -85,B 0,C 180,E1 -30041.01,E2 -30041.01} C_VEL
LIN {X 0,Y 91.528,Z 524.714,A -85,B 0,C 180,E1 -30043.707,E2 -30043.707} C_VEL
LIN {X 0,Y 101.505,Z 518.341,A -85,B 0,C 180,E1 -30045.779,E2 -30045.779} C_VEL
LIN {X 0,Y 111.586,Z 510.4,A -85,B 0,C 180,E1 -30047.489,E2 -30047.489} C_VEL
LIN {X 0,Y 120.063,Z 502.332,A -85,B 0,C 180,E1 -30048.665,E2 -30048.665} C_VEL
LIN {X 0,Y 128.594,Z 492.509,A -85,B 0,C 180,E1 -30049.661,E2 -30049.661} C_VEL
LIN {X 0,Y 135.461,Z 482.874,A -85,B 0,C 180,E1 -30050.323,E2 -30050.323} C_VEL
LIN {X 0,Y 141.494,Z 472.503,A -85,B 0,C 180,E1 -30050.825,E2 -30050.825} C_VEL
LIN {X 0,Y 146.399,Z 461.873,A -85,B 0,C 180,E1 -30051.239,E2 -30051.239} C_VEL
LIN {X 0,Y 146.872,Z 460.58,A -85,B 0,C 180,E1 -30051.4,E2 -30051.4} C_VEL
LIN {X 0,Y 146.79,Z 459.721,A -85,B 0,C 180,E1 -30054.505,E2 -30054.505} C_VEL
LIN {X 0,Y 146.844,Z 459.598,A -85,B 0,C 180,E1 -30057.256,E2 -30057.256} C_VEL
LIN {X 0,Y 146.763,Z 460.405,A -85,B 0,C 180,E1 -30059.314,E2 -30059.314} C_VEL
LIN {X 0,Y 141.369,Z 472.161,A -85,B 0,C 180,E1 -30060,E2 -30060} C_VEL
LIN {X 0,Y 134.425,Z 483.804,A -85,B 0,C 180,E1 -30060.782,E2 -30060.782} C_VEL
LIN {X 0,Y 126.572,Z 494.366,A -85,B 0,C 180,E1 -30061.849,E2 -30061.849} C_VEL
LIN {X 0,Y 117,Z 504.654,A -85,B 0,C 180,E1 -30063.32,E2 -30063.32} C_VEL
LIN {X 0,Y 107.575,Z 512.868,A -85,B 0,C 180,E1 -30064.919,E2 -30064.919} C_VEL
LIN {X 0,Y 97.366,Z 520.137,A -85,B 0,C 180,E1 -30067.016,E2 -30067.016} C_VEL
LIN {X 0,Y 86.685,Z 526.179,A -85,B 0,C 180,E1 -30069.845,E2 -30069.845} C_VEL
LIN {X 0,Y 81.557,Z 528.617,A -85,B 0,C 180,E1 -30070.984,E2 -30070.984} C_VEL
LIN {X 0,Y 72.358,Z 532.133,A -85,B 0,C 180,E1 -30071.925,E2 -30071.925} C_VEL
LIN {X 0,Y 62.942,Z 534.851,A -85,B 0,C 180,E1 -30073.211,E2 -30073.211} C_VEL
LIN {X 0,Y 57.559,Z 536.021,A -85,B 0,C 180,E1 -30075.239,E2 -30075.239} C_VEL
LIN {X 0,Y 51.958,Z 537.091,A -85,B 0,C 180,E1 -30078.756,E2 -30078.756} C_VEL
LIN {X 0,Y 46.031,Z 537.822,A -85,B 0,C 180,E1 -30083.631,E2 -30083.631} C_VEL
LIN {X 0,Y 35.584,Z 538.077,A -85,B 0,C 180,E1 -30097.804,E2 -30097.804} C_VEL
LIN {X 0,Y 31.45,Z 537.614,A -85,B 0,C 180,E1 -30107.893,E2 -30107.893} C_VEL
LIN {X 0,Y 28.459,Z 536.706,A -85,B 0,C 180,E1 -30120.394,E2 -30120.394} C_VEL
LIN {X 0,Y 27.008,Z 535.396,A -85,B 0,C 180,E1 -30134.909,E2 -30134.909} C_VEL
LIN {X 0,Y 28.499,Z 532.273,A -85,B 0,C 180,E1 -30159.464,E2 -30159.464} C_VEL
LIN {X 0,Y 32.269,Z 528.888,A -85,B 0,C 180,E1 -30175.815,E2 -30175.815} C_VEL
LIN {X 0,Y 38.617,Z 524.038,A -85,B 0,C 180,E1 -30189.558,E2 -30189.558} C_VEL
LIN {X 0,Y 46.482,Z 517.921,A -85,B 0,C 180,E1 -30199.104,E2 -30199.104} C_VEL
LIN {X 0,Y 55.125,Z 510.334,A -85,B 0,C 180,E1 -30205.958,E2 -30205.958} C_VEL
LIN {X 0,Y 62.798,Z 502.554,A -85,B 0,C 180,E1 -30210.143,E2 -30210.143} C_VEL
LIN {X 0,Y 70.741,Z 493.043,A -85,B 0,C 180,E1 -30213.39,E2 -30213.39} C_VEL
LIN {X 0,Y 78.001,Z 482.502,A -85,B 0,C 180,E1 -30215.813,E2 -30215.813} C_VEL
LIN {X 0,Y 84.594,Z 470.7,A -85,B 0,C 180,E1 -30217.547,E2 -30217.547} C_VEL
LIN {X 0,Y 89.854,Z 458.154,A -85,B 0,C 180,E1 -30219.01,E2 -30219.01} C_VEL
LIN {X 0,Y 93.682,Z 445.622,A -85,B 0,C 180,E1 -30220.098,E2 -30220.098} C_VEL
LIN {X 0,Y 96.317,Z 433.022,A -85,B 0,C 180,E1 -30220.588,E2 -30220.588} C_VEL
LIN {X 0,Y 97.828,Z 420.781,A -85,B 0,C 180,E1 -30220.973,E2 -30220.973} C_VEL
LIN {X 0,Y 96.902,Z 417.486,A -85,B 0,C 180,E1 -30224.758,E2 -30224.758} C_VEL
LIN {X 0,Y 96.397,Z 415.764,A -85,B 0,C 180,E1 -30227.634,E2 -30227.634} C_VEL
LIN {X 0,Y 96.064,Z 413.73,A -85,B 0,C 180,E1 -30231.587,E2 -30231.587} C_VEL
LIN {X 0,Y 96.134,Z 413.553,A -85,B 0,C 180,E1 -30238.43,E2 -30238.43} C_VEL
LIN {X 0,Y 96.786,Z 416.804,A -85,B 0,C 180,E1 -30244.034,E2 -30244.034} C_VEL
LIN {X 0,Y 97.841,Z 420.709,A -85,B 0,C 180,E1 -30248.534,E2 -30248.534} C_VEL
LIN {X 0,Y 97.535,Z 424.003,A -85,B 0,C 180,E1 -30248.804,E2 -30248.804} C_VEL
LIN {X 0,Y 95.269,Z 439.87,A -85,B 0,C 180,E1 -30249.293,E2 -30249.293} C_VEL
LIN {X 0,Y 92.292,Z 451.97,A -85,B 0,C 180,E1 -30249.894,E2 -30249.894} C_VEL
LIN {X 0,Y 87.649,Z 464.891,A -85,B 0,C 180,E1 -30250.829,E2 -30250.829} C_VEL
LIN {X 0,Y 81.768,Z 477.171,A -85,B 0,C 180,E1 -30252.142,E2 -30252.142} C_VEL
LIN {X 0,Y 75.111,Z 488.103,A -85,B 0,C 180,E1 -30253.904,E2 -30253.904} C_VEL
LIN {X 0,Y 67.761,Z 498.014,A -85,B 0,C 180,E1 -30256.401,E2 -30256.401} C_VEL
LIN {X 0,Y 59.818,Z 507.031,A -85,B 0,C 180,E1 -30259.974,E2 -30259.974} C_VEL
LIN {X 0,Y 51.833,Z 514.564,A -85,B 0,C 180,E1 -30264.28,E2 -30264.28} C_VEL
LIN {X 0,Y 46.279,Z 519.487,A -85,B 0,C 180,E1 -30269.177,E2 -30269.177} C_VEL
LIN {X 0,Y 39.57,Z 524.827,A -85,B 0,C 180,E1 -30276.953,E2 -30276.953} C_VEL
LIN {X 0,Y 32.77,Z 529.985,A -85,B 0,C 180,E1 -30289.963,E2 -30289.963} C_VEL
LIN {X 0,Y 28.413,Z 533.982,A -85,B 0,C 180,E1 -30308.229,E2 -30308.229} C_VEL
LIN {X 0,Y 27.272,Z 536.907,A -85,B 0,C 180,E1 -30330.008,E2 -30330.008} C_VEL
LIN {X 0,Y 27.68,Z 538.239,A -85,B 0,C 180,E1 -30344.716,E2 -30344.716} C_VEL
LIN {X 0,Y 32.942,Z 539.721,A -85,B 0,C 180,E1 -30369.802,E2 -30369.802} C_VEL
LIN {X 0,Y 37.276,Z 539.89,A -85,B 0,C 180,E1 -30378.96,E2 -30378.96} C_VEL
LIN {X 0,Y 48.055,Z 539.016,A -85,B 0,C 180,E1 -30391.348,E2 -30391.348} C_VEL
LIN {X 0,Y 60.24,Z 536.611,A -85,B 0,C 180,E1 -30398.969,E2 -30398.969} C_VEL
LIN {X 0,Y 69.854,Z 533.697,A -85,B 0,C 180,E1 -30402.908,E2 -30402.908} C_VEL
LIN {X 0,Y 79.733,Z 529.781,A -85,B 0,C 180,E1 -30405.841,E2 -30405.841} C_VEL
LIN {X 0,Y 89.796,Z 524.76,A -85,B 0,C 180,E1 -30408.056,E2 -30408.056} C_VEL
LIN {X 0,Y 100,Z 518.48,A -85,B 0,C 180,E1 -30409.718,E2 -30409.718} C_VEL
LIN {X 0,Y 110.269,Z 510.646,A -85,B 0,C 180,E1 -30411.084,E2 -30411.084} C_VEL
LIN {X 0,Y 118.875,Z 502.679,A -85,B 0,C 180,E1 -30412.01,E2 -30412.01} C_VEL
LIN {X 0,Y 127.516,Z 492.977,A -85,B 0,C 180,E1 -30412.783,E2 -30412.783} C_VEL
LIN {X 0,Y 135.315,Z 482.218,A -85,B 0,C 180,E1 -30413.34,E2 -30413.34} C_VEL
LIN {X 0,Y 142.028,Z 470.459,A -85,B 0,C 180,E1 -30413.767,E2 -30413.767} C_VEL
LIN {X 0,Y 143.424,Z 467.634,A -85,B 0,C 180,E1 -30413.847,E2 -30413.847} C_VEL
LIN {X 0,Y 144.002,Z 466.297,A -85,B 0,C 180,E1 -30414.398,E2 -30414.398} C_VEL
LIN {X 0,Y 144.011,Z 466.162,A -85,B 0,C 180,E1 -30416.502,E2 -30416.502} C_VEL
LIN {X 0,Y 143.413,Z 467.455,A -85,B 0,C 180,E1 -30416.849,E2 -30416.849} C_VEL
LIN {X 0,Y 136.924,Z 479.374,A -85,B 0,C 180,E1 -30417.509,E2 -30417.509} C_VEL
LIN {X 0,Y 130.973,Z 488.189,A -85,B 0,C 180,E1 -30418.067,E2 -30418.067} C_VEL
LIN {X 0,Y 123.011,Z 497.933,A -85,B 0,C 180,E1 -30418.991,E2 -30418.991} C_VEL
LIN {X 0,Y 113.759,Z 507.178,A -85,B 0,C 180,E1 -30420.143,E2 -30420.143} C_VEL
LIN {X 0,Y 103.704,Z 515.281,A -85,B 0,C 180,E1 -30421.567,E2 -30421.567} C_VEL
LIN {X 0,Y 93.288,Z 522.086,A -85,B 0,C 180,E1 -30423.402,E2 -30423.402} C_VEL
LIN {X 0,Y 81.295,Z 528.285,A -85,B 0,C 180,E1 -30426.17,E2 -30426.17} C_VEL
LIN {X 0,Y 71.201,Z 532.27,A -85,B 0,C 180,E1 -30429.212,E2 -30429.212} C_VEL
LIN {X 0,Y 61.42,Z 535.17,A -85,B 0,C 180,E1 -30433.229,E2 -30433.229} C_VEL
LIN {X 0,Y 57.559,Z 536.021,A -85,B 0,C 180,E1 -30435.239,E2 -30435.239} C_VEL
LIN {X 0,Y 52.219,Z 537.024,A -85,B 0,C 180,E1 -30437.719,E2 -30437.719} C_VEL
LIN {X 0,Y 42.752,Z 538.081,A -85,B 0,C 180,E1 -30441.081,E2 -30441.081} C_VEL
LIN {X 0,Y 33.436,Z 538.402,A -85,B 0,C 180,E1 -30446.249,E2 -30446.249} C_VEL
LIN {X 0,Y 28.627,Z 538.118,A -85,B 0,C 180,E1 -30452.627,E2 -30452.627} C_VEL
LIN {X 0,Y 22.452,Z 537.078,A -85,B 0,C 180,E1 -30471.229,E2 -30471.229} C_VEL
LIN {X 0,Y 20.127,Z 535.797,A -85,B 0,C 180,E1 -30489.551,E2 -30489.551} C_VEL
LIN {X 0,Y 21.824,Z 532.438,A -85,B 0,C 180,E1 -30524.976,E2 -30524.976} C_VEL
LIN {X 0,Y 28.291,Z 527.97,A -85,B 0,C 180,E1 -30548.381,E2 -30548.381} C_VEL
LIN {X 0,Y 37.746,Z 521.767,A -85,B 0,C 180,E1 -30562.299,E2 -30562.299} C_VEL
LIN {X 0,Y 46.794,Z 515.032,A -85,B 0,C 180,E1 -30569.712,E2 -30569.712} C_VEL
LIN {X 0,Y 56.322,Z 506.669,A -85,B 0,C 180,E1 -30574.769,E2 -30574.769} C_VEL
LIN {X 0,Y 64.518,Z 498.038,A -85,B 0,C 180,E1 -30577.797,E2 -30577.797} C_VEL
LIN {X 0,Y 72.878,Z 487.392,A -85,B 0,C 180,E1 -30580.082,E2 -30580.082} C_VEL
LIN {X 0,Y 79.61,Z 476.817,A -85,B 0,C 180,E1 -30581.613,E2 -30581.613} C_VEL
LIN {X 0,Y 85.491,Z 465.076,A -85,B 0,C 180,E1 -30582.862,E2 -30582.862} C_VEL
LIN {X 0,Y 90.163,Z 452.588,A -85,B 0,C 180,E1 -30583.973,E2 -30583.973} C_VEL
LIN {X 0,Y 93.526,Z 440.072,A -85,B 0,C 180,E1 -30584.582,E2 -30584.582} C_VEL
LIN {X 0,Y 95.789,Z 426.01,A -85,B 0,C 180,E1 -30584.908,E2 -30584.908} C_VEL
LIN {X 0,Y 95.879,Z 424.803,A -85,B 0,C 180,E1 -30585.124,E2 -30585.124} C_VEL
LIN {X 0,Y 95.396,Z 422.732,A -85,B 0,C 180,E1 -30588.312,E2 -30588.312} C_VEL
LIN {X 0,Y 95.128,Z 420.695,A -85,B 0,C 180,E1 -30592.572,E2 -30592.572} C_VEL
LIN {X 0,Y 95.197,Z 420.686,A -85,B 0,C 180,E1 -30597.885,E2 -30597.885} C_VEL
LIN {X 0,Y 95.607,Z 423.428,A -85,B 0,C 180,E1 -30602.634,E2 -30602.634} C_VEL
LIN {X 0,Y 95.932,Z 424.985,A -85,B 0,C 180,E1 -30604.641,E2 -30604.641} C_VEL
